		(* Method outputs *)
		(* Clear output data area *)
		(* Number of output arguments *)
		nNoOfOutputArgs := stRemovePathData.iNoOfOutputArgs;
		(* Set up output argument information *)
		MEMSET(ADR(aOutputArgInfo), 0, SIZEOF(aOutputArgInfo));
		aOutputArgInfo[1].DataType := eUAType_Uint16;
		aOutputArgInfo[1].ValueRank := -1;
		aOutputArgInfo[1].nLenData := SIZEOF(stRemovePathData.stOutput.eStatus);
		aOutputArgInfo[2].DataType := eUAType_String;
		aOutputArgInfo[2].ValueRank := -1;
		aOutputArgInfo[2].nLenData := SIZEOF(stRemovePathData.stOutput.sMessage);
		(* Set up output  *)
		MEMSET(ADR(stRemovePathData.stOutput), 0, SIZEOF(stRemovePathData.stOutput));
		stRemovePathData.stOutput.nNumberOfOutputArguments := nNoOfOutputArgs;
		stRemovePathData.stOutput.stOutputArgInfo[1] := aOutputArgInfo[1];
		stRemovePathData.stOutput.stOutputArgInfo[2] := aOutputArgInfo[2];
	
		(* Execute FB *)
		fbCallMethod.nNumberOfInputArguments := nNoOfInputArgs;
		fbCallMethod.pInputArgInfo := ADR(aInputArgInfo);
		fbCallMethod.cbInputArgInfo := (SIZEOF(aInputArgInfo[1])*nNoOfInputArgs);
		fbCallMethod.pInputArgData := ADR(aInputData);
		fbCallMethod.cbInputArgData := nOffset;
		fbCallMethod.nNumberOfOutputArguments := nNoOfOutputArgs; 
		fbCallMethod.pOutputArgInfo := ADR(aOutputArgInfo); 
		fbCallMethod.cbOutputArgInfo := (SIZEOF(aOutputArgInfo[1]) * nNoOfOutputArgs); 
		fbCallMethod.pOutputArgInfoAndData := ADR(stRemovePathData.stOutput);
		fbCallMethod.cbOutputArgInfoAndData := SIZEOF(stRemovePathData.stOutput);
		
		stRemovePathData.iStatus := 1;
		bCallMethod := TRUE;
		
	ELSIF (stRemovePathData.iStatus = 1) THEN
		// Method call Completed...
		IF (eStateMethod = E_TrackClientState.Connected) THEN
			// Method call OK
			IF (stRemovePathData.stOutput.eStatus = E_MMServerStatus.eMMServerStatus_Success) THEN
				// Method returned OK
				stRemovePathData.iStatus := 2;
			ELSE
				// Method returned with error
				stRemovePathData.iStatus := 3;
				stRemovePathData.stOutput.sMessage;
			END_IF
		ELSIF (eStateMethod = E_TrackClientState.Error) THEN
			// Method call failed
			stRemovePathData.iStatus := 3;
		END_IF
		
	END_IF
END_IF

M_CallRemovePath := stRemovePathData.iStatus;
END_METHOD

METHOD PROTECTED M_CallRemovePathSegment : INT
VAR_INPUT
	iSegmentNo		: UINT;
END_VAR
IF (stRemovePathSegmentData.iStatus = 2) OR (stRemovePathSegmentData.iStatus = 3) THEN
	stRemovePathSegmentData.iStatus := 0;
END_IF

IF (bConnectedMethod AND NOT bBusyMethod) THEN
	IF (stRemovePathSegmentData.iStatus = 0) THEN
	(* Setup method calling parameters *)
		(* Method identifier *)
		sObjectIDentifier := stRemovePathSegmentData.sObjectID;
		sMethodIdentifier := stRemovePathSegmentData.sMethodID;
	
		(* Method Inputs *)
		stRemovePathSegmentData.stInput.sCellID := sCellID;
		stRemovePathSegmentData.stInput.sSegmentID := CONCAT(sCellID, '_PS');
		stRemovePathSegmentData.stInput.sSegmentID := CONCAT(stRemovePathSegmentData.stInput.sSegmentID, UINT_TO_STRING(iSegmentNo));			
		(* Fill input data area with method arguments *)
		MEMSET(ADR(aInputData), 0 ,SIZEOF(aInputData));
		nOffset := 0;
		nOffset := nOffset + MEMCPY(ADR(aInputData)+nOffset, ADR(stRemovePathSegmentData.stInput),	MIN(SIZEOF(stRemovePathSegmentData.stInput), (SIZEOF(aInputData)-nOffset)) );
		(* Number of input arguments *)
		nNoOfInputArgs := stRemovePathSegmentData.iNoOfInputArgs;
		(* Set up input argument information *)
		MEMSET(ADR(aInputArgInfo), 0, SIZEOF(aInputArgInfo));
		aInputArgInfo[1].DataType := eUAType_String;
		aInputArgInfo[1].ValueRank := -1;	// -1: Scalar 
		aInputArgInfo[1].nLenData := SIZEOF(stRemovePathSegmentData.stInput.sCellID);
		aInputArgInfo[2].DataType := eUAType_String;
		aInputArgInfo[2].ValueRank := -1;	// -1: Scalar 
		aInputArgInfo[2].nLenData := SIZEOF(stRemovePathSegmentData.stInput.sSegmentID);
		
		(* Method outputs *)
		(* Clear output data area *)
		(* Number of output arguments *)
		nNoOfOutputArgs := stRemovePathSegmentData.iNoOfOutputArgs;
		(* Set up output argument information *)
		MEMSET(ADR(aOutputArgInfo), 0, SIZEOF(aOutputArgInfo));
		aOutputArgInfo[1].DataType := eUAType_Uint16;
		aOutputArgInfo[1].ValueRank := -1;
		aOutputArgInfo[1].nLenData := SIZEOF(stRemovePathSegmentData.stOutput.eStatus);
		aOutputArgInfo[2].DataType := eUAType_String;
		aOutputArgInfo[2].ValueRank := -1;
		aOutputArgInfo[2].nLenData := SIZEOF(stRemovePathSegmentData.stOutput.sMessage);
		(* Set up output  *)
		MEMSET(ADR(stRemovePathSegmentData.stOutput), 0, SIZEOF(stRemovePathSegmentData.stOutput));
		stRemovePathSegmentData.stOutput.nNumberOfOutputArguments := nNoOfOutputArgs;
		stRemovePathSegmentData.stOutput.stOutputArgInfo[1] := aOutputArgInfo[1];
		stRemovePathSegmentData.stOutput.stOutputArgInfo[2] := aOutputArgInfo[2];
	
		(* Execute FB *)
		fbCallMethod.nNumberOfInputArguments := nNoOfInputArgs;
		fbCallMethod.pInputArgInfo := ADR(aInputArgInfo);
		fbCallMethod.cbInputArgInfo := (SIZEOF(aInputArgInfo[1])*nNoOfInputArgs);
		fbCallMethod.pInputArgData := ADR(aInputData);
		fbCallMethod.cbInputArgData := nOffset;
		fbCallMethod.nNumberOfOutputArguments := nNoOfOutputArgs; 
		fbCallMethod.pOutputArgInfo := ADR(aOutputArgInfo); 
		fbCallMethod.cbOutputArgInfo := (SIZEOF(aOutputArgInfo[1]) * nNoOfOutputArgs); 
		fbCallMethod.pOutputArgInfoAndData := ADR(stRemovePathSegmentData.stOutput);
		fbCallMethod.cbOutputArgInfoAndData := SIZEOF(stRemovePathSegmentData.stOutput);
		
		stRemovePathSegmentData.iStatus := 1;
		bCallMethod := TRUE;
		
	ELSIF (stRemovePathSegmentData.iStatus = 1) THEN
		// Method call Completed...
		IF (eStateMethod = E_TrackClientState.Connected) THEN
			// Method call OK
			IF (stRemovePathSegmentData.stOutput.eStatus = E_MMServerStatus.eMMServerStatus_Success) THEN
				// Method returned OK
				stRemovePathSegmentData.iStatus := 2;
			ELSE
				// Method returned with error
				stRemovePathSegmentData.iStatus := 3;
				stRemovePathSegmentData.stOutput.sMessage;
			END_IF
		ELSIF (eStateMethod = E_TrackClientState.Error) THEN
			// Method call failed
			stRemovePathSegmentData.iStatus := 3;
		END_IF
		
	END_IF
END_IF

M_CallRemovePathSegment := stRemovePathSegmentData.iStatus;
END_METHOD

METHOD PROTECTED M_CallRemoveReservation : INT
VAR_INPUT
	sStationID					: STRING(30);												(* The identifier for the station. *)
	nTicket						: UINT;														(*  *)
END_VAR
VAR
	i					: UINT;	
END_VAR
IF (stRemoveReservationData.iStatus = 2) OR (stRemoveReservationData.iStatus = 3) THEN
	stRemoveReservationData.iStatus := 0;
END_IF

IF (bConnectedMethod AND NOT bBusyMethod) THEN
	IF (stRemoveReservationData.iStatus = 0) THEN
	(* Setup method calling parameters *)
		(* Method identifier *)
		sObjectIDentifier := stRemoveReservationData.sObjectID;
		sMethodIdentifier := stRemoveReservationData.sMethodID;
	
		(* Method Inputs *)
		stRemoveReservationData.stInput.sStationID := sStationID;
		stRemoveReservationData.stInput.nTicket := nTicket;
		(* Fill input data area with method arguments *)
		MEMSET(ADR(aInputData), 0 ,SIZEOF(aInputData));
		nOffset := 0;
		nOffset := nOffset + MEMCPY(ADR(aInputData)+nOffset, ADR(stRemoveReservationData.stInput),	MIN(SIZEOF(stRemoveReservationData.stInput), (SIZEOF(aInputData)-nOffset)) );
		(* Number of input arguments *)
		nNoOfInputArgs := stRemoveReservationData.iNoOfInputArgs;
		(* Set up input argument information *)
		MEMSET(ADR(aInputArgInfo), 0, SIZEOF(aInputArgInfo));
		aInputArgInfo[1].DataType := eUAType_String;
		aInputArgInfo[1].ValueRank := -1;	// -1: Scalar 
		aInputArgInfo[1].nLenData := SIZEOF(stRemoveReservationData.stInput.sStationID);
		aInputArgInfo[2].DataType := eUAType_UInt16;
		aInputArgInfo[2].ValueRank := -1;	// -1: Scalar 
		aInputArgInfo[2].nLenData := SIZEOF(stRemoveReservationData.stInput.nTicket);
		
		(* Method outputs *)
		(* Clear output data area *)
		(* Number of output arguments *)
		nNoOfOutputArgs := stRemoveReservationData.iNoOfOutputArgs;
		(* Set up output argument information *)
		MEMSET(ADR(aOutputArgInfo), 0, SIZEOF(aOutputArgInfo));
		aOutputArgInfo[1].DataType := eUAType_Uint16;
		aOutputArgInfo[1].ValueRank := -1;
		aOutputArgInfo[1].nLenData := SIZEOF(stRemoveReservationData.stOutput.eStatus);
		aOutputArgInfo[2].DataType := eUAType_String;
		aOutputArgInfo[2].ValueRank := -1;
		aOutputArgInfo[2].nLenData := SIZEOF(stRemoveReservationData.stOutput.sMessage);
		(* Set up output  *)
		MEMSET(ADR(stRemoveReservationData.stOutput), 0, SIZEOF(stRemoveReservationData.stOutput));
		stRemoveReservationData.stOutput.nNumberOfOutputArguments := nNoOfOutputArgs;
		stRemoveReservationData.stOutput.stOutputArgInfo[1] := aOutputArgInfo[1];
		stRemoveReservationData.stOutput.stOutputArgInfo[2] := aOutputArgInfo[2];
	
		(* Execute FB *)
		fbCallMethod.nNumberOfInputArguments := nNoOfInputArgs;
		fbCallMethod.pInputArgInfo := ADR(aInputArgInfo);
		fbCallMethod.cbInputArgInfo := (SIZEOF(aInputArgInfo[1])*nNoOfInputArgs);
		fbCallMethod.pInputArgData := ADR(aInputData);
		fbCallMethod.cbInputArgData := nOffset;
		fbCallMethod.nNumberOfOutputArguments := nNoOfOutputArgs; 
		fbCallMethod.pOutputArgInfo := ADR(aOutputArgInfo); 
		fbCallMethod.cbOutputArgInfo := (SIZEOF(aOutputArgInfo[1]) * nNoOfOutputArgs); 
		fbCallMethod.pOutputArgInfoAndData := ADR(stRemoveReservationData.stOutput);
		fbCallMethod.cbOutputArgInfoAndData := SIZEOF(stRemoveReservationData.stOutput);
		
		stRemoveReservationData.iStatus := 1;
		bCallMethod := TRUE;
		
	ELSIF (stRemoveReservationData.iStatus = 1) THEN
		// Method call Completed...
		IF (eStateMethod = E_TrackClientState.Connected) THEN
			// Method call OK
			IF (stRemoveReservationData.stOutput.eStatus = E_MMServerStatus.eMMServerStatus_Success) THEN
				// Method returned OK
				stRemoveReservationData.iStatus := 2;
			ELSE
				// Method returned with error
				stRemoveReservationData.iStatus := 3;
				stRemoveReservationData.stOutput.sMessage;
			END_IF
		ELSIF (eStateMethod = E_TrackClientState.Error) THEN
			// Method call failed
			stRemoveReservationData.iStatus := 3;
		END_IF
		
	END_IF
END_IF

M_CallRemoveReservation := stRemoveReservationData.iStatus;
END_METHOD

METHOD PROTECTED M_CallRemoveStation : INT
VAR_INPUT
	nStationNo			: UINT(1..5);
END_VAR
IF (stRemoveStationData.iStatus = 2) OR (stRemoveStationData.iStatus = 3) THEN
	stRemoveStationData.iStatus := 0;
END_IF

IF (bConnectedMethod AND NOT bBusyMethod) THEN
	IF (stRemoveStationData.iStatus = 0) THEN
	(* Setup method calling parameters *)
		(* Method identifier *)
		sObjectIDentifier := stRemoveStationData.sObjectID;
		sMethodIdentifier := stRemoveStationData.sMethodID;
	
		(* Method Inputs *)
		stRemoveStationData.stInput.sCellID := sCellID;
		stRemoveStationData.stInput.sStationID := aStations[nStationNo].sStationID;
		(* Fill input data area with method arguments *)
		MEMSET(ADR(aInputData), 0 ,SIZEOF(aInputData));
		nOffset := 0;
		nOffset := nOffset + MEMCPY(ADR(aInputData)+nOffset, ADR(stRemoveStationData.stInput),	MIN(SIZEOF(stRemoveStationData.stInput), (SIZEOF(aInputData)-nOffset)) );
		(* Number of input arguments *)
		nNoOfInputArgs := stRemoveStationData.iNoOfInputArgs;
		(* Set up input argument information *)
		MEMSET(ADR(aInputArgInfo), 0, SIZEOF(aInputArgInfo));
		aInputArgInfo[1].DataType := eUAType_String;
		aInputArgInfo[1].ValueRank := -1;	// -1: Scalar 
		aInputArgInfo[1].nLenData := SIZEOF(stRemoveStationData.stInput.sCellID);
		aInputArgInfo[2].DataType := eUAType_String;
		aInputArgInfo[2].ValueRank := -1;	// -1: Scalar 
		aInputArgInfo[2].nLenData := SIZEOF(stRemoveStationData.stInput.sStationID);
		
		(* Method outputs *)
		(* Clear output data area *)
		(* Number of output arguments *)
		nNoOfOutputArgs := stRemoveStationData.iNoOfOutputArgs;
		(* Set up output argument information *)
		MEMSET(ADR(aOutputArgInfo), 0, SIZEOF(aOutputArgInfo));
		aOutputArgInfo[1].DataType := eUAType_Uint16;
		aOutputArgInfo[1].ValueRank := -1;
		aOutputArgInfo[1].nLenData := SIZEOF(stRemoveStationData.stOutput.eStatus);
		aOutputArgInfo[2].DataType := eUAType_String;
		aOutputArgInfo[2].ValueRank := -1;
		aOutputArgInfo[2].nLenData := SIZEOF(stRemoveStationData.stOutput.sMessage);
		(* Set up output  *)
		MEMSET(ADR(stRemoveStationData.stOutput), 0, SIZEOF(stRemoveStationData.stOutput));
		stRemoveStationData.stOutput.nNumberOfOutputArguments := nNoOfOutputArgs;
		stRemoveStationData.stOutput.stOutputArgInfo[1] := aOutputArgInfo[1];
		stRemoveStationData.stOutput.stOutputArgInfo[2] := aOutputArgInfo[2];
	
		(* Execute FB *)
		fbCallMethod.nNumberOfInputArguments := nNoOfInputArgs;
		fbCallMethod.pInputArgInfo := ADR(aInputArgInfo);
		fbCallMethod.cbInputArgInfo := (SIZEOF(aInputArgInfo[1])*nNoOfInputArgs);
		fbCallMethod.pInputArgData := ADR(aInputData);
		fbCallMethod.cbInputArgData := nOffset;
		fbCallMethod.nNumberOfOutputArguments := nNoOfOutputArgs; 
		fbCallMethod.pOutputArgInfo := ADR(aOutputArgInfo); 
		fbCallMethod.cbOutputArgInfo := (SIZEOF(aOutputArgInfo[1]) * nNoOfOutputArgs); 
		fbCallMethod.pOutputArgInfoAndData := ADR(stRemoveStationData.stOutput);
		fbCallMethod.cbOutputArgInfoAndData := SIZEOF(stRemoveStationData.stOutput);
		
		stRemoveStationData.iStatus := 1;
		bCallMethod := TRUE;
		
	ELSIF (stRemoveStationData.iStatus = 1) THEN
		// Method call Completed...
		IF (eStateMethod = E_TrackClientState.Connected) THEN
			// Method call OK
			IF (stRemoveStationData.stOutput.eStatus = E_MMServerStatus.eMMServerStatus_Success) THEN
				// Method returned OK
				stRemoveStationData.iStatus := 2;
			ELSE
				// Method returned with error
				stRemoveStationData.iStatus := 3;
				stRemoveStationData.stOutput.sMessage;
			END_IF
		ELSIF (eStateMethod = E_TrackClientState.Error) THEN
			// Method call failed
			stRemoveStationData.iStatus := 3;
		END_IF
		
	END_IF
END_IF

M_CallRemoveStation := stRemoveStationData.iStatus;
END_METHOD

METHOD PROTECTED M_CallRemoveTrafficLight : INT
VAR_INPUT
END_VAR
IF (stRemoveTrafficLightData.iStatus = 2) OR (stRemoveTrafficLightData.iStatus = 3) THEN
	stRemoveTrafficLightData.iStatus := 0;
END_IF

IF (bConnectedMethod AND NOT bBusyMethod) THEN
	IF (stRemoveTrafficLightData.iStatus = 0) THEN
	(* Setup method calling parameters *)
		(* Method identifier *)
		sObjectIDentifier := stRemoveTrafficLightData.sObjectID;
		sMethodIdentifier := stRemoveTrafficLightData.sMethodID;
	
		(* Method Inputs *)
		stRemoveTrafficLightData.stInput.sCellID := sCellID;
		stRemoveTrafficLightData.stInput.sID := CONCAT(sCellID, '_TL');
		(* Fill input data area with method arguments *)
		MEMSET(ADR(aInputData), 0 ,SIZEOF(aInputData));
		nOffset := 0;
		nOffset := nOffset + MEMCPY(ADR(aInputData)+nOffset, ADR(stRemoveTrafficLightData.stInput),	MIN(SIZEOF(stRemoveTrafficLightData.stInput),	(SIZEOF(aInputData)-nOffset)) );
		(* Number of input arguments *)
		nNoOfInputArgs := stRemoveTrafficLightData.iNoOfInputArgs;
		(* Set up input argument information *)
		MEMSET(ADR(aInputArgInfo), 0, SIZEOF(aInputArgInfo));
		aInputArgInfo[1].DataType := eUAType_String;
		aInputArgInfo[1].ValueRank := -1;	// -1: Scalar 
		aInputArgInfo[1].nLenData := SIZEOF(stRemoveTrafficLightData.stInput.sCellID);
		aInputArgInfo[2].DataType := eUAType_String;
		aInputArgInfo[2].ValueRank := -1;	// -1: Scalar 
		aInputArgInfo[2].nLenData := SIZEOF(stRemoveTrafficLightData.stInput.sID);
		
		(* Method outputs *)
		(* Clear output data area *)
		(* Number of output arguments *)
		nNoOfOutputArgs := stRemoveTrafficLightData.iNoOfOutputArgs;
		(* Set up output argument information *)
		MEMSET(ADR(aOutputArgInfo), 0, SIZEOF(aOutputArgInfo));
		aOutputArgInfo[1].DataType := eUAType_Uint16;
		aOutputArgInfo[1].ValueRank := -1;
		aOutputArgInfo[1].nLenData := SIZEOF(stRemoveTrafficLightData.stOutput.eStatus);
		aOutputArgInfo[2].DataType := eUAType_String;
		aOutputArgInfo[2].ValueRank := -1;
		aOutputArgInfo[2].nLenData := SIZEOF(stRemoveTrafficLightData.stOutput.sMessage);
		(* Set up output  *)
		MEMSET(ADR(stRemoveTrafficLightData.stOutput), 0, SIZEOF(stRemoveTrafficLightData.stOutput));
		stRemoveTrafficLightData.stOutput.nNumberOfOutputArguments := nNoOfOutputArgs;
		stRemoveTrafficLightData.stOutput.stOutputArgInfo[1] := aOutputArgInfo[1];
		stRemoveTrafficLightData.stOutput.stOutputArgInfo[2] := aOutputArgInfo[2];
	
		(* Execute FB *)
		fbCallMethod.nNumberOfInputArguments := nNoOfInputArgs;
		fbCallMethod.pInputArgInfo := ADR(aInputArgInfo);
		fbCallMethod.cbInputArgInfo := (SIZEOF(aInputArgInfo[1])*nNoOfInputArgs);
		fbCallMethod.pInputArgData := ADR(aInputData);
		fbCallMethod.cbInputArgData := nOffset;
		fbCallMethod.nNumberOfOutputArguments := nNoOfOutputArgs; 
		fbCallMethod.pOutputArgInfo := ADR(aOutputArgInfo); 
		fbCallMethod.cbOutputArgInfo := (SIZEOF(aOutputArgInfo[1]) * nNoOfOutputArgs); 
		fbCallMethod.pOutputArgInfoAndData := ADR(stRemoveTrafficLightData.stOutput);
		fbCallMethod.cbOutputArgInfoAndData := SIZEOF(stRemoveTrafficLightData.stOutput);
		
		stRemoveTrafficLightData.iStatus := 1;
		bCallMethod := TRUE;
		
	ELSIF (stRemoveTrafficLightData.iStatus = 1) THEN
		// Method call Completed...
		IF (eStateMethod = E_TrackClientState.Connected) THEN
			// Method call OK
			IF (stRemoveTrafficLightData.stOutput.eStatus = E_MMServerStatus.eMMServerStatus_Success) THEN
				// Method returned OK
				stRemoveTrafficLightData.iStatus := 2;
			ELSE
				// Method returned with error
				stRemoveTrafficLightData.iStatus := 3;
				stRemoveTrafficLightData.stOutput.sMessage;
			END_IF
		ELSIF (eStateMethod = E_TrackClientState.Error) THEN
			// Method call failed
			stRemoveTrafficLightData.iStatus := 3;
		END_IF
		
	END_IF
END_IF

M_CallRemoveTrafficLight := stRemoveTrafficLightData.iStatus;
END_METHOD

METHOD PROTECTED M_CallResetPath : INT
VAR_INPUT
	nPathNo			: UINT(1..5);
END_VAR
IF (stResetPathData.iStatus = 2) OR (stResetPathData.iStatus = 3) THEN
	stResetPathData.iStatus := 0;
END_IF

IF (bConnectedMethod AND NOT bBusyMethod) THEN
	IF (stResetPathData.iStatus = 0) THEN
	(* Setup method calling parameters *)
		(* Method identifier *)
		sObjectIDentifier := stResetPathData.sObjectID;
		sMethodIdentifier := stResetPathData.sMethodID;
	
		(* Method Inputs *)
		stResetPathData.stInput.iPath := nPathNo;
		(* Fill input data area with method arguments *)
		MEMSET(ADR(aInputData), 0 ,SIZEOF(aInputData));
		nOffset := 0;
		nOffset := nOffset + MEMCPY(ADR(aInputData)+nOffset, ADR(stResetPathData.stInput),	MIN(SIZEOF(stResetPathData.stInput), (SIZEOF(aInputData)-nOffset)) );
		(* Number of input arguments *)
		nNoOfInputArgs := stResetPathData.iNoOfInputArgs;
		(* Set up input argument information *)
		MEMSET(ADR(aInputArgInfo), 0, SIZEOF(aInputArgInfo));
		aInputArgInfo[1].DataType := eUAType_UInt16;
		aInputArgInfo[1].ValueRank := -1;	// -1: Scalar 
		aInputArgInfo[1].nLenData := SIZEOF(stResetPathData.stInput.iPath);
		
		(* Method outputs *)
		(* Clear output data area *)
		(* Number of output arguments *)
		nNoOfOutputArgs := stResetPathData.iNoOfOutputArgs;
		(* Set up output argument information *)
		MEMSET(ADR(aOutputArgInfo), 0, SIZEOF(aOutputArgInfo));
		aOutputArgInfo[1].DataType := eUAType_Uint16;
		aOutputArgInfo[1].ValueRank := -1;
		aOutputArgInfo[1].nLenData := SIZEOF(stResetPathData.stOutput.eStatus);
		aOutputArgInfo[2].DataType := eUAType_String;
		aOutputArgInfo[2].ValueRank := -1;
		aOutputArgInfo[2].nLenData := SIZEOF(stResetPathData.stOutput.sMessage);
		(* Set up output  *)
		MEMSET(ADR(stResetPathData.stOutput), 0, SIZEOF(stResetPathData.stOutput));
		stResetPathData.stOutput.nNumberOfOutputArguments := nNoOfOutputArgs;
		stResetPathData.stOutput.stOutputArgInfo[1] := aOutputArgInfo[1];
		stResetPathData.stOutput.stOutputArgInfo[2] := aOutputArgInfo[2];
	
		(* Execute FB *)
		fbCallMethod.nNumberOfInputArguments := nNoOfInputArgs;
		fbCallMethod.pInputArgInfo := ADR(aInputArgInfo);
		fbCallMethod.cbInputArgInfo := (SIZEOF(aInputArgInfo[1])*nNoOfInputArgs);
		fbCallMethod.pInputArgData := ADR(aInputData);
		fbCallMethod.cbInputArgData := nOffset;
		fbCallMethod.nNumberOfOutputArguments := nNoOfOutputArgs; 
		fbCallMethod.pOutputArgInfo := ADR(aOutputArgInfo); 
		fbCallMethod.cbOutputArgInfo := (SIZEOF(aOutputArgInfo[1]) * nNoOfOutputArgs); 
		fbCallMethod.pOutputArgInfoAndData := ADR(stResetPathData.stOutput);
		fbCallMethod.cbOutputArgInfoAndData := SIZEOF(stResetPathData.stOutput);
		
		stResetPathData.iStatus := 1;
		bCallMethod := TRUE;
		
	ELSIF (stResetPathData.iStatus = 1) THEN
		// Method call Completed...
		IF (eStateMethod = E_TrackClientState.Connected) THEN
			// eStateMethod call OK
			IF (stResetPathData.stOutput.eStatus = E_MMServerStatus.eMMServerStatus_Success) THEN
				// Method returned OK
				stResetPathData.iStatus := 2;
			ELSE
				// Method returned with error
				stResetPathData.iStatus := 3;
				stResetPathData.stOutput.sMessage;
			END_IF
		ELSIF (eStateMethod = E_TrackClientState.Error) THEN
			// Method call failed
			stResetPathData.iStatus := 3;
		END_IF
		
	END_IF
END_IF

M_CallResetPath := stResetPathData.iStatus;
END_METHOD

METHOD PROTECTED M_CallResumePath : INT
VAR_INPUT
	nPathNo			: UINT(1..5);
END_VAR
IF (stResumePathData.iStatus = 2) OR (stResumePathData.iStatus = 3) THEN
	stResumePathData.iStatus := 0;
END_IF

IF (bConnectedMethod AND NOT bBusyMethod) THEN
	IF (stResumePathData.iStatus = 0) THEN
	(* Setup method calling parameters *)
		(* Method identifier *)
		sObjectIDentifier := stResumePathData.sObjectID;
		sMethodIdentifier := stResumePathData.sMethodID;
	
		(* Method Inputs *)
		stResumePathData.stInput.iPath := nPathNo;
		(* Fill input data area with method arguments *)
		MEMSET(ADR(aInputData), 0 ,SIZEOF(aInputData));
		nOffset := 0;
		nOffset := nOffset + MEMCPY(ADR(aInputData)+nOffset, ADR(stResumePathData.stInput),	MIN(SIZEOF(stResumePathData.stInput), (SIZEOF(aInputData)-nOffset)) );
		(* Number of input arguments *)
		nNoOfInputArgs := stResumePathData.iNoOfInputArgs;
		(* Set up input argument information *)
		MEMSET(ADR(aInputArgInfo), 0, SIZEOF(aInputArgInfo));
		aInputArgInfo[1].DataType := eUAType_UInt16;
		aInputArgInfo[1].ValueRank := -1;	// -1: Scalar 
		aInputArgInfo[1].nLenData := SIZEOF(stResumePathData.stInput.iPath);
		
		(* Method outputs *)
		(* Clear output data area *)
		(* Number of output arguments *)
		nNoOfOutputArgs := stResumePathData.iNoOfOutputArgs;
		(* Set up output argument information *)
		MEMSET(ADR(aOutputArgInfo), 0, SIZEOF(aOutputArgInfo));
		aOutputArgInfo[1].DataType := eUAType_Uint16;
		aOutputArgInfo[1].ValueRank := -1;
		aOutputArgInfo[1].nLenData := SIZEOF(stResumePathData.stOutput.eStatus);
		aOutputArgInfo[2].DataType := eUAType_String;
		aOutputArgInfo[2].ValueRank := -1;
		aOutputArgInfo[2].nLenData := SIZEOF(stResumePathData.stOutput.sMessage);
		(* Set up output  *)
		MEMSET(ADR(stResumePathData.stOutput), 0, SIZEOF(stResumePathData.stOutput));
		stResumePathData.stOutput.nNumberOfOutputArguments := nNoOfOutputArgs;
		stResumePathData.stOutput.stOutputArgInfo[1] := aOutputArgInfo[1];
		stResumePathData.stOutput.stOutputArgInfo[2] := aOutputArgInfo[2];
	
		(* Execute FB *)
		fbCallMethod.nNumberOfInputArguments := nNoOfInputArgs;
		fbCallMethod.pInputArgInfo := ADR(aInputArgInfo);
		fbCallMethod.cbInputArgInfo := (SIZEOF(aInputArgInfo[1])*nNoOfInputArgs);
		fbCallMethod.pInputArgData := ADR(aInputData);
		fbCallMethod.cbInputArgData := nOffset;
		fbCallMethod.nNumberOfOutputArguments := nNoOfOutputArgs; 
		fbCallMethod.pOutputArgInfo := ADR(aOutputArgInfo); 
		fbCallMethod.cbOutputArgInfo := (SIZEOF(aOutputArgInfo[1]) * nNoOfOutputArgs); 
		fbCallMethod.pOutputArgInfoAndData := ADR(stResumePathData.stOutput);
		fbCallMethod.cbOutputArgInfoAndData := SIZEOF(stResumePathData.stOutput);
		
		stResumePathData.iStatus := 1;
		bCallMethod := TRUE;
		
	ELSIF (stResumePathData.iStatus = 1) THEN
		// Method call Completed...
		IF (eStateMethod = E_TrackClientState.Connected) THEN
			// Method call OK
			IF (stResumePathData.stOutput.eStatus = E_MMServerStatus.eMMServerStatus_Success) THEN
				// Method returned OK
				stResumePathData.iStatus := 2;
			ELSE
				// Method returned with error
				stResumePathData.iStatus := 3;
				stResumePathData.stOutput.sMessage;
			END_IF
		ELSIF (eStateMethod = E_TrackClientState.Error) THEN
			// Method call failed
			stResumePathData.iStatus := 3;
		END_IF
		
	END_IF
END_IF

M_CallResumePath := stResumePathData.iStatus;
END_METHOD

METHOD PROTECTED M_CallSetTrafficLightColor : INT
VAR_INPUT
	nTrafficLightNo	: UINT;
	nColor			: INT;
END_VAR
IF (stSetTrafficLightColorData.iStatus = 2) OR (stSetTrafficLightColorData.iStatus = 3) THEN
	stSetTrafficLightColorData.iStatus := 0;
END_IF

IF (bConnectedMethod AND NOT bBusyMethod) THEN
	IF (stSetTrafficLightColorData.iStatus = 0) THEN
	(* Setup method calling parameters *)
		(* Method identifier *)
		sObjectIDentifier := stSetTrafficLightColorData.sObjectID;
		sMethodIdentifier := stSetTrafficLightColorData.sMethodID;
			
		(* Method Inputs *)
		stSetTrafficLightColorData.stInput.sCellID := sCellID;
		stSetTrafficLightColorData.stInput.sID := CONCAT(sCellID, '_TL');
		stSetTrafficLightColorData.stInput.sID := CONCAT(stSetTrafficLightColorData.stInput.sID, UINT_TO_STRING(nTrafficLightNo));
		stSetTrafficLightColorData.stInput.nColor := nColor;
		(* Fill input data area with method arguments *)
		MEMSET(ADR(aInputData), 0 ,SIZEOF(aInputData));
		nOffset := 0;
		nOffset := nOffset + MEMCPY(ADR(aInputData)+nOffset, ADR(stSetTrafficLightColorData.stInput),	MIN(SIZEOF(stSetTrafficLightColorData.stInput),	(SIZEOF(aInputData)-nOffset)) );
		(* Number of input arguments *)
		nNoOfInputArgs := stSetTrafficLightColorData.iNoOfInputArgs;
		(* Set up input argument information *)
		MEMSET(ADR(aInputArgInfo), 0, SIZEOF(aInputArgInfo));
		aInputArgInfo[1].DataType := eUAType_String;
		aInputArgInfo[1].ValueRank := -1;	// -1: Scalar 
		aInputArgInfo[1].nLenData := SIZEOF(stSetTrafficLightColorData.stInput.sCellID);
		aInputArgInfo[2].DataType := eUAType_String;
		aInputArgInfo[2].ValueRank := -1;	// -1: Scalar 
		aInputArgInfo[2].nLenData := SIZEOF(stSetTrafficLightColorData.stInput.sID);
		aInputArgInfo[3].DataType := eUAType_Int16;
		aInputArgInfo[3].ValueRank := -1;	// -1: Scalar 
		aInputArgInfo[3].nLenData := SIZEOF(nColor);
		
		(* Method outputs *)
		(* Clear output data area *)
		(* Number of output arguments *)
		nNoOfOutputArgs := stSetTrafficLightColorData.iNoOfOutputArgs;
		(* Set up output argument information *)
		MEMSET(ADR(aOutputArgInfo), 0, SIZEOF(aOutputArgInfo));
		aOutputArgInfo[1].DataType := eUAType_Uint16;
		aOutputArgInfo[1].ValueRank := -1;
		aOutputArgInfo[1].nLenData := SIZEOF(stSetTrafficLightColorData.stOutput.eStatus);
		aOutputArgInfo[2].DataType := eUAType_String;
		aOutputArgInfo[2].ValueRank := -1;
		aOutputArgInfo[2].nLenData := SIZEOF(stSetTrafficLightColorData.stOutput.sMessage);
		(* Set up output  *)
		MEMSET(ADR(stSetTrafficLightColorData.stOutput), 0, SIZEOF(stSetTrafficLightColorData.stOutput));
		stSetTrafficLightColorData.stOutput.nNumberOfOutputArguments := nNoOfOutputArgs;
		stSetTrafficLightColorData.stOutput.stOutputArgInfo[1] := aOutputArgInfo[1];
		stSetTrafficLightColorData.stOutput.stOutputArgInfo[2] := aOutputArgInfo[2];
	
		(* Execute FB *)
		fbCallMethod.nNumberOfInputArguments := nNoOfInputArgs;
		fbCallMethod.pInputArgInfo := ADR(aInputArgInfo);
		fbCallMethod.cbInputArgInfo := (SIZEOF(aInputArgInfo[1])*nNoOfInputArgs);
		fbCallMethod.pInputArgData := ADR(aInputData);
		fbCallMethod.cbInputArgData := nOffset;
		fbCallMethod.nNumberOfOutputArguments := nNoOfOutputArgs; 
		fbCallMethod.pOutputArgInfo := ADR(aOutputArgInfo); 
		fbCallMethod.cbOutputArgInfo := (SIZEOF(aOutputArgInfo[1]) * nNoOfOutputArgs); 
		fbCallMethod.pOutputArgInfoAndData := ADR(stSetTrafficLightColorData.stOutput);
		fbCallMethod.cbOutputArgInfoAndData := SIZEOF(stSetTrafficLightColorData.stOutput);
		
		stSetTrafficLightColorData.iStatus := 1;
		bCallMethod := TRUE;
		
	ELSIF (stSetTrafficLightColorData.iStatus = 1) THEN
		// Method call Completed...
		IF (eStateMethod = E_TrackClientState.Connected) THEN
			// Method call OK
			IF (stSetTrafficLightColorData.stOutput.eStatus = E_MMServerStatus.eMMServerStatus_Success) THEN
				// Method returned OK
				stSetTrafficLightColorData.iStatus := 2;
			ELSE
				// Method returned with error
				stSetTrafficLightColorData.iStatus := 3;
				stSetTrafficLightColorData.stOutput.sMessage;
			END_IF
		ELSIF (eStateMethod = E_TrackClientState.Error) THEN
			// Method call failed
			stSetTrafficLightColorData.iStatus := 3;
		END_IF
		
	END_IF
END_IF

M_CallSetTrafficLightColor := stSetTrafficLightColorData.iStatus;
END_METHOD

METHOD PROTECTED M_CallStartPath : INT
VAR_INPUT
	nPathNo			: UINT(1..5);
END_VAR
IF (stStartPathData.iStatus = 2) OR (stStartPathData.iStatus = 3) THEN
	stStartPathData.iStatus := 0;
END_IF

IF (bConnectedMethod AND NOT bBusyMethod) THEN
	IF (stStartPathData.iStatus = 0) THEN
	(* Setup method calling parameters *)
		(* Method identifier *)
		sObjectIDentifier := stStartPathData.sObjectID;
		sMethodIdentifier := stStartPathData.sMethodID;
	
		(* Method Inputs *)
		stStartPathData.stInput.iPath := nPathNo;
		(* Fill input data area with method arguments *)
		MEMSET(ADR(aInputData), 0 ,SIZEOF(aInputData));
		nOffset := 0;
		nOffset := nOffset + MEMCPY(ADR(aInputData)+nOffset, ADR(stStartPathData.stInput),	MIN(SIZEOF(stStartPathData.stInput), (SIZEOF(aInputData)-nOffset)) );
		(* Number of input arguments *)
		nNoOfInputArgs := stStartPathData.iNoOfInputArgs;
		(* Set up input argument information *)
		MEMSET(ADR(aInputArgInfo), 0, SIZEOF(aInputArgInfo));
		aInputArgInfo[1].DataType := eUAType_UInt16;
		aInputArgInfo[1].ValueRank := -1;	// -1: Scalar 
		aInputArgInfo[1].nLenData := SIZEOF(stStartPathData.stInput.iPath);
		
		(* Method outputs *)
		(* Clear output data area *)
		(* Number of output arguments *)
		nNoOfOutputArgs := stStartPathData.iNoOfOutputArgs;
		(* Set up output argument information *)
		MEMSET(ADR(aOutputArgInfo), 0, SIZEOF(aOutputArgInfo));
		aOutputArgInfo[1].DataType := eUAType_Uint16;
		aOutputArgInfo[1].ValueRank := -1;
		aOutputArgInfo[1].nLenData := SIZEOF(stStartPathData.stOutput.eStatus);
		aOutputArgInfo[2].DataType := eUAType_String;
		aOutputArgInfo[2].ValueRank := -1;
		aOutputArgInfo[2].nLenData := SIZEOF(stStartPathData.stOutput.sMessage);
		(* Set up output  *)
		MEMSET(ADR(stStartPathData.stOutput), 0, SIZEOF(stStartPathData.stOutput));
		stStartPathData.stOutput.nNumberOfOutputArguments := nNoOfOutputArgs;
		stStartPathData.stOutput.stOutputArgInfo[1] := aOutputArgInfo[1];
		stStartPathData.stOutput.stOutputArgInfo[2] := aOutputArgInfo[2];
	
		(* Execute FB *)
		fbCallMethod.nNumberOfInputArguments := nNoOfInputArgs;
		fbCallMethod.pInputArgInfo := ADR(aInputArgInfo);
		fbCallMethod.cbInputArgInfo := (SIZEOF(aInputArgInfo[1])*nNoOfInputArgs);
		fbCallMethod.pInputArgData := ADR(aInputData);
		fbCallMethod.cbInputArgData := nOffset;
		fbCallMethod.nNumberOfOutputArguments := nNoOfOutputArgs; 
		fbCallMethod.pOutputArgInfo := ADR(aOutputArgInfo); 
		fbCallMethod.cbOutputArgInfo := (SIZEOF(aOutputArgInfo[1]) * nNoOfOutputArgs); 
		fbCallMethod.pOutputArgInfoAndData := ADR(stStartPathData.stOutput);
		fbCallMethod.cbOutputArgInfoAndData := SIZEOF(stStartPathData.stOutput);
		
		stStartPathData.iStatus := 1;
		bCallMethod := TRUE;
		
	ELSIF (stStartPathData.iStatus = 1) THEN
		// Method call Completed...
		IF (eStateMethod = E_TrackClientState.Connected) THEN
			// Method call OK
			IF (stStartPathData.stOutput.eStatus = E_MMServerStatus.eMMServerStatus_Success) THEN
				// Method returned OK
				stStartPathData.iStatus := 2;
			ELSE
				// Method returned with error
				stStartPathData.iStatus := 3;
				stStartPathData.stOutput.sMessage;
			END_IF
		ELSIF (eStateMethod = E_TrackClientState.Error) THEN
			// Method call failed
			stStartPathData.iStatus := 3;
		END_IF
		
	END_IF
END_IF

M_CallStartPath := stStartPathData.iStatus;
END_METHOD

METHOD PROTECTED M_CallSuspendPath : INT
VAR_INPUT
	nPathNo			: UINT(1..5);
END_VAR
IF (stSuspendPathData.iStatus = 2) OR (stSuspendPathData.iStatus = 3) THEN
	stSuspendPathData.iStatus := 0;
END_IF

IF (bConnectedMethod AND NOT bBusyMethod) THEN
	IF (stSuspendPathData.iStatus = 0) THEN
	(* Setup method calling parameters *)
		(* Method identifier *)
		sObjectIDentifier := stSuspendPathData.sObjectID;
		sMethodIdentifier := stSuspendPathData.sMethodID;
	
		(* Method Inputs *)
		stSuspendPathData.stInput.iPath := nPathNo;
		(* Fill input data area with method arguments *)
		MEMSET(ADR(aInputData), 0 ,SIZEOF(aInputData));
		nOffset := 0;
		nOffset := nOffset + MEMCPY(ADR(aInputData)+nOffset, ADR(stSuspendPathData.stInput),	MIN(SIZEOF(stSuspendPathData.stInput), (SIZEOF(aInputData)-nOffset)) );
		(* Number of input arguments *)
		nNoOfInputArgs := stSuspendPathData.iNoOfInputArgs;
		(* Set up input argument information *)
		MEMSET(ADR(aInputArgInfo), 0, SIZEOF(aInputArgInfo));
		aInputArgInfo[1].DataType := eUAType_UInt16;
		aInputArgInfo[1].ValueRank := -1;	// -1: Scalar 
		aInputArgInfo[1].nLenData := SIZEOF(stSuspendPathData.stInput.iPath);
		
		(* Method outputs *)
		(* Clear output data area *)
		(* Number of output arguments *)
		nNoOfOutputArgs := stSuspendPathData.iNoOfOutputArgs;
		(* Set up output argument information *)
		MEMSET(ADR(aOutputArgInfo), 0, SIZEOF(aOutputArgInfo));
		aOutputArgInfo[1].DataType := eUAType_Uint16;
		aOutputArgInfo[1].ValueRank := -1;
		aOutputArgInfo[1].nLenData := SIZEOF(stSuspendPathData.stOutput.eStatus);
		aOutputArgInfo[2].DataType := eUAType_String;
		aOutputArgInfo[2].ValueRank := -1;
		aOutputArgInfo[2].nLenData := SIZEOF(stSuspendPathData.stOutput.sMessage);
		(* Set up output  *)
		MEMSET(ADR(stSuspendPathData.stOutput), 0, SIZEOF(stSuspendPathData.stOutput));
		stSuspendPathData.stOutput.nNumberOfOutputArguments := nNoOfOutputArgs;
		stSuspendPathData.stOutput.stOutputArgInfo[1] := aOutputArgInfo[1];
		stSuspendPathData.stOutput.stOutputArgInfo[2] := aOutputArgInfo[2];
	
		(* Execute FB *)
		fbCallMethod.nNumberOfInputArguments := nNoOfInputArgs;
		fbCallMethod.pInputArgInfo := ADR(aInputArgInfo);
		fbCallMethod.cbInputArgInfo := (SIZEOF(aInputArgInfo[1])*nNoOfInputArgs);
		fbCallMethod.pInputArgData := ADR(aInputData);
		fbCallMethod.cbInputArgData := nOffset;
		fbCallMethod.nNumberOfOutputArguments := nNoOfOutputArgs; 
		fbCallMethod.pOutputArgInfo := ADR(aOutputArgInfo); 
		fbCallMethod.cbOutputArgInfo := (SIZEOF(aOutputArgInfo[1]) * nNoOfOutputArgs); 
		fbCallMethod.pOutputArgInfoAndData := ADR(stSuspendPathData.stOutput);
		fbCallMethod.cbOutputArgInfoAndData := SIZEOF(stSuspendPathData.stOutput);
		
		stSuspendPathData.iStatus := 1;
		bCallMethod := TRUE;
		
	ELSIF (stSuspendPathData.iStatus = 1) THEN
		// Method call Completed...
		IF (eStateMethod = E_TrackClientState.Connected) THEN
			// Method call OK
			IF (stSuspendPathData.stOutput.eStatus = E_MMServerStatus.eMMServerStatus_Success) THEN
				// Method returned OK
				stSuspendPathData.iStatus := 2;
			ELSE
				// Method returned with error
				stSuspendPathData.iStatus := 3;
				stSuspendPathData.stOutput.sMessage;
			END_IF
		ELSIF (eStateMethod = E_TrackClientState.Error) THEN
			// Method call failed
			stSuspendPathData.iStatus := 3;
		END_IF
		
	END_IF
END_IF

M_CallSuspendPath := stSuspendPathData.iStatus;
END_METHOD

METHOD PROTECTED M_CallTrafficLightColor : INT
VAR_INPUT
END_VAR
IF (stTrafficLightColorData.iStatus = 2) OR (stTrafficLightColorData.iStatus = 3) THEN
	stTrafficLightColorData.iStatus := 0;
END_IF

IF (bConnectedMethod AND NOT bBusyMethod) THEN
	IF (stTrafficLightColorData.iStatus = 0) THEN
	(* Setup method calling parameters *)
		(* Method identifier *)
		sObjectIDentifier := stTrafficLightColorData.sObjectID;
		sMethodIdentifier := stTrafficLightColorData.sMethodID;
	
		(* Method Inputs *)
		stTrafficLightColorData.stInput.sCellID := sCellID;
		stTrafficLightColorData.stInput.sID := CONCAT(sCellID, '_TL');
		(* Fill input data area with method arguments *)
		MEMSET(ADR(aInputData), 0 ,SIZEOF(aInputData));
		nOffset := 0;
		nOffset := nOffset + MEMCPY(ADR(aInputData)+nOffset, ADR(stTrafficLightColorData.stInput),	MIN(SIZEOF(stTrafficLightColorData.stInput), (SIZEOF(aInputData)-nOffset)) );
		(* Number of input arguments *)
		nNoOfInputArgs := stTrafficLightColorData.iNoOfInputArgs;
		(* Set up input argument information *)
		MEMSET(ADR(aInputArgInfo), 0, SIZEOF(aInputArgInfo));
		aInputArgInfo[1].DataType := eUAType_String;
		aInputArgInfo[1].ValueRank := -1;	// -1: Scalar 
		aInputArgInfo[1].nLenData := SIZEOF(stTrafficLightColorData.stInput.sCellID);
		aInputArgInfo[2].DataType := eUAType_String;
		aInputArgInfo[2].ValueRank := -1;	// -1: Scalar 
		aInputArgInfo[2].nLenData := SIZEOF(stTrafficLightColorData.stInput.sID);
		
		(* Method outputs *)
		(* Clear output data area *)
		(* Number of output arguments *)
		nNoOfOutputArgs := stTrafficLightColorData.iNoOfOutputArgs;
		(* Set up output argument information *)
		MEMSET(ADR(aOutputArgInfo), 0, SIZEOF(aOutputArgInfo));
		aOutputArgInfo[1].DataType := eUAType_Uint16;
		aOutputArgInfo[1].ValueRank := -1;
		aOutputArgInfo[1].nLenData := SIZEOF(stTrafficLightColorData.stOutput.eStatus);
		aOutputArgInfo[2].DataType := eUAType_String;
		aOutputArgInfo[2].ValueRank := -1;
		aOutputArgInfo[2].nLenData := SIZEOF(stTrafficLightColorData.stOutput.sMessage);
		aOutputArgInfo[3].DataType := eUAType_Int16;
		aOutputArgInfo[3].ValueRank := -1;
		aOutputArgInfo[3].nLenData := SIZEOF(stTrafficLightColorData.stOutput.nTrafficLightColor);
		(* Set up output  *)
		MEMSET(ADR(stTrafficLightColorData.stOutput), 0, SIZEOF(stTrafficLightColorData.stOutput));
		stTrafficLightColorData.stOutput.nNumberOfOutputArguments := nNoOfOutputArgs;
		stTrafficLightColorData.stOutput.stOutputArgInfo[1] := aOutputArgInfo[1];
		stTrafficLightColorData.stOutput.stOutputArgInfo[2] := aOutputArgInfo[2];
		stTrafficLightColorData.stOutput.stOutputArgInfo[3] := aOutputArgInfo[3];
	
		(* Execute FB *)
		fbCallMethod.nNumberOfInputArguments := nNoOfInputArgs;
		fbCallMethod.pInputArgInfo := ADR(aInputArgInfo);
		fbCallMethod.cbInputArgInfo := (SIZEOF(aInputArgInfo[1])*nNoOfInputArgs);
		fbCallMethod.pInputArgData := ADR(aInputData);
		fbCallMethod.cbInputArgData := nOffset;
		fbCallMethod.nNumberOfOutputArguments := nNoOfOutputArgs; 
		fbCallMethod.pOutputArgInfo := ADR(aOutputArgInfo); 
		fbCallMethod.cbOutputArgInfo := (SIZEOF(aOutputArgInfo[1]) * nNoOfOutputArgs); 
		fbCallMethod.pOutputArgInfoAndData := ADR(stTrafficLightColorData.stOutput);
		fbCallMethod.cbOutputArgInfoAndData := SIZEOF(stTrafficLightColorData.stOutput);
		
		stTrafficLightColorData.iStatus := 1;
		bCallMethod := TRUE;
		
	ELSIF (stTrafficLightColorData.iStatus = 1) THEN
		// Method call Completed...
		IF (eStateMethod = E_TrackClientState.Connected) THEN
			// Method call OK
			IF (stTrafficLightColorData.stOutput.eStatus = E_MMServerStatus.eMMServerStatus_Success) THEN
				// Method returned OK
				stTrafficLightColorData.iStatus := 2;
			ELSE
				// Method returned with error
				stTrafficLightColorData.iStatus := 3;
				stTrafficLightColorData.stOutput.sMessage;
				stTrafficLightColorData.stOutput.nTrafficLightColor;
			END_IF
		ELSIF (eStateMethod = E_TrackClientState.Error) THEN
			// Method call failed
			stTrafficLightColorData.iStatus := 3;
		END_IF
		
	END_IF
END_IF

M_CallTrafficLightColor := stTrafficLightColorData.iStatus;
END_METHOD

METHOD PROTECTED M_CallUpdateStationBuffer : INT
VAR_INPUT
	sStationID			: STRING(30);
	eBufferType			: E_MMStationBuffer;
	nBufferIndex		: USINT;	
	nVehicleID			: UINT;
	sCarrierID			: STRING(30);
	nTicket				: UINT;
	nPriority			: UINT;
END_VAR
VAR
END_VAR
IF (stUpdateStationBufferData.iStatus = 2) OR (stUpdateStationBufferData.iStatus = 3) THEN
	stUpdateStationBufferData.iStatus := 0;
END_IF

IF (bConnectedMethod AND NOT bBusyMethod) THEN
	IF (stUpdateStationBufferData.iStatus = 0) THEN
	(* Setup method calling parameters *)
		(* Method identifier *)
		sObjectIDentifier := stUpdateStationBufferData.sObjectID;
		sMethodIdentifier := stUpdateStationBufferData.sMethodID;
	
		(* Method Inputs *)
		stUpdateStationBufferData.stInput.sStationID := sStationID;
		stUpdateStationBufferData.stInput.eStationBufferType := eBufferType;
		stUpdateStationBufferData.stInput.nIndex := nBufferIndex;
		stUpdateStationBufferData.stInput.nVehicleID := nVehicleID;
		stUpdateStationBufferData.stInput.sCarrierID := sCarrierID;
		stUpdateStationBufferData.stInput.nTicket := nTicket;
		stUpdateStationBufferData.stInput.nPriority := nPriority;
		
		(* Fill input data area with method arguments *)
		MEMSET(ADR(aInputData), 0 ,SIZEOF(aInputData));
		nOffset := 0;
		nOffset := nOffset + MEMCPY(ADR(aInputData)+nOffset, ADR(stUpdateStationBufferData.stInput),	MIN(SIZEOF(stUpdateStationBufferData.stInput), (SIZEOF(aInputData)-nOffset)) );
		(* Number of input arguments *)
		nNoOfInputArgs := stUpdateStationBufferData.iNoOfInputArgs;
		(* Set up input argument information *)
		MEMSET(ADR(aInputArgInfo), 0, SIZEOF(aInputArgInfo));
		aInputArgInfo[1].DataType := eUAType_String;
		aInputArgInfo[1].ValueRank := -1;	// -1: Scalar 
		aInputArgInfo[1].nLenData := SIZEOF(stUpdateStationBufferData.stInput.sStationID);
		aInputArgInfo[2].DataType := eUAType_UInt16;
		aInputArgInfo[2].ValueRank := -1;	// -1: Scalar 
		aInputArgInfo[2].nLenData := SIZEOF(stUpdateStationBufferData.stInput.eStationBufferType);
		aInputArgInfo[3].DataType := eUAType_Byte;
		aInputArgInfo[3].ValueRank := -1;	// -1: Scalar 
		aInputArgInfo[3].nLenData := SIZEOF(stUpdateStationBufferData.stInput.nIndex);
		aInputArgInfo[4].DataType := eUAType_UInt16;
		aInputArgInfo[4].ValueRank := -1;	// -1: Scalar 
		aInputArgInfo[4].nLenData := SIZEOF(stUpdateStationBufferData.stInput.nVehicleID);
		aInputArgInfo[5].DataType := eUAType_String;
		aInputArgInfo[5].ValueRank := -1;	// -1: Scalar 
		aInputArgInfo[5].nLenData := SIZEOF(stUpdateStationBufferData.stInput.sCarrierID);
		aInputArgInfo[6].DataType := eUAType_UInt16;
		aInputArgInfo[6].ValueRank := -1;	// -1: Scalar 
		aInputArgInfo[6].nLenData := SIZEOF(stUpdateStationBufferData.stInput.nTicket);
		aInputArgInfo[7].DataType := eUAType_UInt16;
		aInputArgInfo[7].ValueRank := -1;	// -1: Scalar 
		aInputArgInfo[7].nLenData := SIZEOF(stUpdateStationBufferData.stInput.nPriority);
		
		(* Method outputs *)
		(* Clear output data area *)
		(* Number of output arguments *)
		nNoOfOutputArgs := stUpdateStationBufferData.iNoOfOutputArgs;
		(* Set up output argument information *)
		MEMSET(ADR(aOutputArgInfo), 0, SIZEOF(aOutputArgInfo));
		aOutputArgInfo[1].DataType := eUAType_Uint16;
		aOutputArgInfo[1].ValueRank := -1;
		aOutputArgInfo[1].nLenData := SIZEOF(stUpdateStationBufferData.stOutput.eStatus);
		aOutputArgInfo[2].DataType := eUAType_String;
		aOutputArgInfo[2].ValueRank := -1;
		aOutputArgInfo[2].nLenData := SIZEOF(stUpdateStationBufferData.stOutput.sMessage);
		(* Set up output  *)
		MEMSET(ADR(stUpdateStationBufferData.stOutput), 0, SIZEOF(stUpdateStationBufferData.stOutput));
		stUpdateStationBufferData.stOutput.nNumberOfOutputArguments := nNoOfOutputArgs;
		stUpdateStationBufferData.stOutput.stOutputArgInfo[1] := aOutputArgInfo[1];
		stUpdateStationBufferData.stOutput.stOutputArgInfo[2] := aOutputArgInfo[2];
	
		(* Execute FB *)
		fbCallMethod.nNumberOfInputArguments := nNoOfInputArgs;
		fbCallMethod.pInputArgInfo := ADR(aInputArgInfo);
		fbCallMethod.cbInputArgInfo := (SIZEOF(aInputArgInfo[1])*nNoOfInputArgs);
		fbCallMethod.pInputArgData := ADR(aInputData);
		fbCallMethod.cbInputArgData := nOffset;
		fbCallMethod.nNumberOfOutputArguments := nNoOfOutputArgs; 
		fbCallMethod.pOutputArgInfo := ADR(aOutputArgInfo); 
		fbCallMethod.cbOutputArgInfo := (SIZEOF(aOutputArgInfo[1]) * nNoOfOutputArgs); 
		fbCallMethod.pOutputArgInfoAndData := ADR(stUpdateStationBufferData.stOutput);
		fbCallMethod.cbOutputArgInfoAndData := SIZEOF(stUpdateStationBufferData.stOutput);
		
		stUpdateStationBufferData.iStatus := 1;
		bCallMethod := TRUE;
		
	ELSIF (stUpdateStationBufferData.iStatus = 1) THEN
		// Method call Completed...
		IF (eStateMethod = E_TrackClientState.Connected) THEN
			// Method call OK
			IF (stUpdateStationBufferData.stOutput.eStatus = E_MMServerStatus.eMMServerStatus_Success) THEN
				// Method returned OK
				stUpdateStationBufferData.iStatus := 2;
			ELSE
				// Method returned with error
				stUpdateStationBufferData.iStatus := 3;
				stUpdateStationBufferData.stOutput.sMessage;
			END_IF
		ELSIF (eStateMethod = E_TrackClientState.Error) THEN
			// Method call failed
			stUpdateStationBufferData.iStatus := 3;
		END_IF
		
	END_IF
ELSE
	M_CallUpdateStationBuffer := -1;
	RETURN;
END_IF

M_CallUpdateStationBuffer := stUpdateStationBufferData.iStatus;
END_METHOD

METHOD M_CallUpdateVehicleMappingData : INT
VAR_INPUT
	nVehicleID			: UINT;										(* Magnemotion Vehicle ID *)
	sCarrierID			: STRING(30);								(* Carrier ID *)
	bTool				: BOOL;										(*  *)
	sToolID				: STRING(30);								(* Tool ID *)
	bMaterial			: BOOL;										(*  *)
	sMaterialID			: STRING(30);								(* Material ID string *)
END_VAR
VAR
END_VAR
IF (stUpdateVehicleMappingDataData.iStatus = 2) OR (stUpdateVehicleMappingDataData.iStatus = 3) THEN
	stUpdateVehicleMappingDataData.iStatus := 0;
END_IF

IF (bConnectedMethod AND NOT bBusyMethod) THEN
	IF (stUpdateVehicleMappingDataData.iStatus = 0) THEN
	(* Setup method calling parameters *)
		(* Method identifier *)
		sObjectIDentifier := stUpdateVehicleMappingDataData.sObjectID;
		sMethodIdentifier := stUpdateVehicleMappingDataData.sMethodID;
	
		(* Method Inputs *)
		stUpdateVehicleMappingDataData.stInput.nVehicleID := nVehicleID;
		stUpdateVehicleMappingDataData.stInput.sCarrierID := sCarrierID;
		stUpdateVehicleMappingDataData.stInput.bTool := bTool;
		stUpdateVehicleMappingDataData.stInput.sToolID := sToolID;
		stUpdateVehicleMappingDataData.stInput.bMaterial := bMaterial;
		stUpdateVehicleMappingDataData.stInput.sMaterialID := sMaterialID;
		
		(* Fill input data area with method arguments *)
		MEMSET(ADR(aInputData), 0 ,SIZEOF(aInputData));
		nOffset := 0;
		nOffset := nOffset + MEMCPY(ADR(aInputData)+nOffset, ADR(stUpdateVehicleMappingDataData.stInput),	MIN(SIZEOF(stUpdateVehicleMappingDataData.stInput), (SIZEOF(aInputData)-nOffset)) );
		(* Number of input arguments *)
		nNoOfInputArgs := stUpdateVehicleMappingDataData.iNoOfInputArgs;
		(* Set up input argument information *)
		MEMSET(ADR(aInputArgInfo), 0, SIZEOF(aInputArgInfo));
		aInputArgInfo[1].DataType := eUAType_UInt16;
		aInputArgInfo[1].ValueRank := -1;	// -1: Scalar 
		aInputArgInfo[1].nLenData := SIZEOF(stUpdateVehicleMappingDataData.stInput.nVehicleID);
		aInputArgInfo[2].DataType := eUAType_String;
		aInputArgInfo[2].ValueRank := -1;	// -1: Scalar 
		aInputArgInfo[2].nLenData := SIZEOF(stUpdateVehicleMappingDataData.stInput.sCarrierID);
		aInputArgInfo[3].DataType := eUAType_Boolean;
		aInputArgInfo[3].ValueRank := -1;	// -1: Scalar 
		aInputArgInfo[3].nLenData := SIZEOF(stUpdateVehicleMappingDataData.stInput.bTool);
		aInputArgInfo[4].DataType := eUAType_String;
		aInputArgInfo[4].ValueRank := -1;	// -1: Scalar 
		aInputArgInfo[4].nLenData := SIZEOF(stUpdateVehicleMappingDataData.stInput.sToolID);
		aInputArgInfo[5].DataType := eUAType_Boolean;
		aInputArgInfo[5].ValueRank := -1;	// -1: Scalar 
		aInputArgInfo[5].nLenData := SIZEOF(stUpdateVehicleMappingDataData.stInput.bMaterial);
		aInputArgInfo[6].DataType := eUAType_String;
		aInputArgInfo[6].ValueRank := -1;	// -1: Scalar 
		aInputArgInfo[6].nLenData := SIZEOF(stUpdateVehicleMappingDataData.stInput.sMaterialID);
		
		(* Method outputs *)
		(* Clear output data area *)
		(* Number of output arguments *)
		nNoOfOutputArgs := stUpdateVehicleMappingDataData.iNoOfOutputArgs;
		(* Set up output argument information *)
		MEMSET(ADR(aOutputArgInfo), 0, SIZEOF(aOutputArgInfo));
		aOutputArgInfo[1].DataType := eUAType_Uint16;
		aOutputArgInfo[1].ValueRank := -1;
		aOutputArgInfo[1].nLenData := SIZEOF(stUpdateVehicleMappingDataData.stOutput.eStatus);
		aOutputArgInfo[2].DataType := eUAType_String;
		aOutputArgInfo[2].ValueRank := -1;
		aOutputArgInfo[2].nLenData := SIZEOF(stUpdateVehicleMappingDataData.stOutput.sMessage);
		(* Set up output  *)
		MEMSET(ADR(stUpdateVehicleMappingDataData.stOutput), 0, SIZEOF(stUpdateVehicleMappingDataData.stOutput));
		stUpdateVehicleMappingDataData.stOutput.nNumberOfOutputArguments := nNoOfOutputArgs;
		stUpdateVehicleMappingDataData.stOutput.stOutputArgInfo[1] := aOutputArgInfo[1];
		stUpdateVehicleMappingDataData.stOutput.stOutputArgInfo[2] := aOutputArgInfo[2];
	
		(* Execute FB *)
		fbCallMethod.nNumberOfInputArguments := nNoOfInputArgs;
		fbCallMethod.pInputArgInfo := ADR(aInputArgInfo);
		fbCallMethod.cbInputArgInfo := (SIZEOF(aInputArgInfo[1])*nNoOfInputArgs);
		fbCallMethod.pInputArgData := ADR(aInputData);
		fbCallMethod.cbInputArgData := nOffset;
		fbCallMethod.nNumberOfOutputArguments := nNoOfOutputArgs; 
		fbCallMethod.pOutputArgInfo := ADR(aOutputArgInfo); 
		fbCallMethod.cbOutputArgInfo := (SIZEOF(aOutputArgInfo[1]) * nNoOfOutputArgs); 
		fbCallMethod.pOutputArgInfoAndData := ADR(stUpdateVehicleMappingDataData.stOutput);
		fbCallMethod.cbOutputArgInfoAndData := SIZEOF(stUpdateVehicleMappingDataData.stOutput);
		
		stUpdateVehicleMappingDataData.iStatus := 1;
		bCallMethod := TRUE;
		
	ELSIF (stUpdateVehicleMappingDataData.iStatus = 1) THEN
		// Method call Completed...
		IF (eStateMethod = E_TrackClientState.Connected) THEN
			// Method call OK
			IF (stUpdateVehicleMappingDataData.stOutput.eStatus = E_MMServerStatus.eMMServerStatus_Success) THEN
				// Method returned OK
				stUpdateVehicleMappingDataData.iStatus := 2;
				// Trig vehicle data reading because data has changed
				M_VehicleToReadAdd(stUpdateVehicleMappingDataData.stInput.nVehicleID);
				
			ELSE
				// Method returned with error
				stUpdateVehicleMappingDataData.iStatus := 3;
				stUpdateVehicleMappingDataData.stOutput.sMessage;
				
			END_IF
			
		ELSIF (eStateMethod = E_TrackClientState.Error) THEN
			// Method call failed
			stUpdateVehicleMappingDataData.iStatus := 3;
			
		END_IF
		
	END_IF
ELSE
	M_CallUpdateVehicleMappingData := -1;
	RETURN;
	
END_IF

M_CallUpdateVehicleMappingData := stUpdateVehicleMappingDataData.iStatus;
END_METHOD

METHOD M_CallUpdateVehicleMontage : INT
VAR_INPUT
	nVehicleID			: UINT;										(* Magnemotion Vehicle ID *)
	bTool				: BOOL;										(*  *)
	sToolID				: STRING(30);								(* Tool ID *)
	bMaterial			: BOOL;										(*  *)
	sMaterialID			: STRING(30);								(* Material ID string *)
	bReserved			: BOOL;										(* TRUE signals vehicle is reserved for montage line *)
END_VAR
VAR
END_VAR
IF (stUpdateVehicleMontageData.iStatus = 2) OR (stUpdateVehicleMontageData.iStatus = 3) THEN
	stUpdateVehicleMontageData.iStatus := 0;
END_IF

IF (bConnectedMethod AND NOT bBusyMethod) THEN
	IF (stUpdateVehicleMontageData.iStatus = 0) THEN
	(* Setup method calling parameters *)
		(* Method identifier *)
		sObjectIDentifier := stUpdateVehicleMontageData.sObjectID;
		sMethodIdentifier := stUpdateVehicleMontageData.sMethodID;
	
		(* Method Inputs *)
		stUpdateVehicleMontageData.stInput.eInputType := E_MMVehicleInputType.eMMVehicleInputType_VehicleID;
		stUpdateVehicleMontageData.stInput.sInput := UINT_TO_STRING(nVehicleID);
		stUpdateVehicleMontageData.stInput.bTool := bTool;
		stUpdateVehicleMontageData.stInput.sToolID := sToolID;
		stUpdateVehicleMontageData.stInput.bMaterial := bMaterial;
		stUpdateVehicleMontageData.stInput.sMaterialID := sMaterialID;
		stUpdateVehicleMontageData.stInput.bReserved := bReserved;
		
		(* Fill input data area with method arguments *)
		MEMSET(ADR(aInputData), 0 ,SIZEOF(aInputData));
		nOffset := 0;
		nOffset := nOffset + MEMCPY(ADR(aInputData)+nOffset, ADR(stUpdateVehicleMontageData.stInput),	MIN(SIZEOF(stUpdateVehicleMontageData.stInput), (SIZEOF(aInputData)-nOffset)) );
		(* Number of input arguments *)
		nNoOfInputArgs := stUpdateVehicleMontageData.iNoOfInputArgs;
		(* Set up input argument information *)
		MEMSET(ADR(aInputArgInfo), 0, SIZEOF(aInputArgInfo));
		aInputArgInfo[1].DataType := eUAType_UInt16;
		aInputArgInfo[1].ValueRank := -1;	// -1: Scalar 
		aInputArgInfo[1].nLenData := SIZEOF(stUpdateVehicleMontageData.stInput.eInputType);
		aInputArgInfo[2].DataType := eUAType_String;
		aInputArgInfo[2].ValueRank := -1;	// -1: Scalar 
		aInputArgInfo[2].nLenData := SIZEOF(stUpdateVehicleMontageData.stInput.sInput);
		aInputArgInfo[3].DataType := eUAType_Boolean;
		aInputArgInfo[3].ValueRank := -1;	// -1: Scalar 
		aInputArgInfo[3].nLenData := SIZEOF(stUpdateVehicleMontageData.stInput.bTool);
		aInputArgInfo[4].DataType := eUAType_String;
		aInputArgInfo[4].ValueRank := -1;	// -1: Scalar 
		aInputArgInfo[4].nLenData := SIZEOF(stUpdateVehicleMontageData.stInput.sToolID);
		aInputArgInfo[5].DataType := eUAType_Boolean;
		aInputArgInfo[5].ValueRank := -1;	// -1: Scalar 
		aInputArgInfo[5].nLenData := SIZEOF(stUpdateVehicleMontageData.stInput.bMaterial);
		aInputArgInfo[6].DataType := eUAType_String;
		aInputArgInfo[6].ValueRank := -1;	// -1: Scalar 
		aInputArgInfo[6].nLenData := SIZEOF(stUpdateVehicleMontageData.stInput.sMaterialID);
		aInputArgInfo[7].DataType := eUAType_Boolean;
		aInputArgInfo[7].ValueRank := -1;	// -1: Scalar 
		aInputArgInfo[7].nLenData := SIZEOF(stUpdateVehicleMontageData.stInput.bReserved);
		
		(* Method outputs *)
		(* Clear output data area *)
		(* Number of output arguments *)
		nNoOfOutputArgs := stUpdateVehicleMontageData.iNoOfOutputArgs;
		(* Set up output argument information *)
		MEMSET(ADR(aOutputArgInfo), 0, SIZEOF(aOutputArgInfo));
		aOutputArgInfo[1].DataType := eUAType_Uint16;
		aOutputArgInfo[1].ValueRank := -1;
		aOutputArgInfo[1].nLenData := SIZEOF(stUpdateVehicleMontageData.stOutput.eStatus);
		aOutputArgInfo[2].DataType := eUAType_String;
		aOutputArgInfo[2].ValueRank := -1;
		aOutputArgInfo[2].nLenData := SIZEOF(stUpdateVehicleMontageData.stOutput.sMessage);
		(* Set up output  *)
		MEMSET(ADR(stUpdateVehicleMontageData.stOutput), 0, SIZEOF(stUpdateVehicleMontageData.stOutput));
		stUpdateVehicleMontageData.stOutput.nNumberOfOutputArguments := nNoOfOutputArgs;
		stUpdateVehicleMontageData.stOutput.stOutputArgInfo[1] := aOutputArgInfo[1];
		stUpdateVehicleMontageData.stOutput.stOutputArgInfo[2] := aOutputArgInfo[2];
	
		(* Execute FB *)
		fbCallMethod.nNumberOfInputArguments := nNoOfInputArgs;
		fbCallMethod.pInputArgInfo := ADR(aInputArgInfo);
		fbCallMethod.cbInputArgInfo := (SIZEOF(aInputArgInfo[1])*nNoOfInputArgs);
		fbCallMethod.pInputArgData := ADR(aInputData);
		fbCallMethod.cbInputArgData := nOffset;
		fbCallMethod.nNumberOfOutputArguments := nNoOfOutputArgs; 
		fbCallMethod.pOutputArgInfo := ADR(aOutputArgInfo); 
		fbCallMethod.cbOutputArgInfo := (SIZEOF(aOutputArgInfo[1]) * nNoOfOutputArgs); 
		fbCallMethod.pOutputArgInfoAndData := ADR(stUpdateVehicleMontageData.stOutput);
		fbCallMethod.cbOutputArgInfoAndData := SIZEOF(stUpdateVehicleMontageData.stOutput);
		
		stUpdateVehicleMontageData.iStatus := 1;
		bCallMethod := TRUE;
		
	ELSIF (stUpdateVehicleMontageData.iStatus = 1) THEN
		// Method call Completed...
		IF (UINT_TO_STRING(nVehicleID) = stUpdateVehicleMontageData.stInput.sInput) THEN
			IF (eStateMethod = E_TrackClientState.Connected) THEN
				// Method call OK
				IF (stUpdateVehicleMontageData.stOutput.eStatus = E_MMServerStatus.eMMServerStatus_Success) THEN
					// Method returned OK
					stUpdateVehicleMontageData.iStatus := 2;
					// Trig vehicle data reading because data has changed
					M_VehicleToReadAdd(nVehicleID);
									
				ELSE
					// Method returned with error
					stUpdateVehicleMontageData.iStatus := 3;
					stUpdateVehicleMontageData.stOutput.sMessage;
					
				END_IF
				
			ELSIF (eStateMethod = E_TrackClientState.Error) THEN
				// Method call failed
				stUpdateVehicleMontageData.iStatus := 3;
	
			END_IF
		ELSE
			// Wrong vehicle ID
			F_LogLine('TC_VMD: Wrong Vehicle ID (%d)', nVehicleID);
			
		END_IF
	END_IF
ELSE
	M_CallUpdateVehicleMontage := -1;
	RETURN;

END_IF

M_CallUpdateVehicleMontage := stUpdateVehicleMontageData.iStatus;
END_METHOD

METHOD PROTECTED M_CallUpdateVehicleOwner : INT
VAR_INPUT
	nVehicleID			: UINT;										(* Magnemotion Vehicle ID *)
	eInputType			: E_MMVehicleInputType;
	sInput				: STRING(30);
	sCellID				: STRING(30);
END_VAR
VAR
END_VAR
IF (stUpdateVehicleOwnerData.iStatus = 2) OR (stUpdateVehicleOwnerData.iStatus = 3) THEN
	stUpdateVehicleOwnerData.iStatus := 0;
END_IF

IF (bConnectedMethod AND NOT bBusyMethod) THEN
	IF (stUpdateVehicleOwnerData.iStatus = 0) THEN
	(* Setup method calling parameters *)
		(* Method identifier *)
		sObjectIDentifier := stUpdateVehicleOwnerData.sObjectID;
		sMethodIdentifier := stUpdateVehicleOwnerData.sMethodID;
	
		(* Method Inputs *)
		stUpdateVehicleOwnerData.stInput.eInputType := eInputType;
		stUpdateVehicleOwnerData.stInput.sInput := sInput;
		stUpdateVehicleOwnerData.stInput.sCellID := sCellID;
		
		(* Fill input data area with method arguments *)
		MEMSET(ADR(aInputData), 0 ,SIZEOF(aInputData));
		nOffset := 0;
		nOffset := nOffset + MEMCPY(ADR(aInputData)+nOffset, ADR(stUpdateVehicleOwnerData.stInput),	MIN(SIZEOF(stUpdateVehicleOwnerData.stInput), (SIZEOF(aInputData)-nOffset)) );
		(* Number of input arguments *)
		nNoOfInputArgs := stUpdateVehicleOwnerData.iNoOfInputArgs;
		(* Set up input argument information *)
		MEMSET(ADR(aInputArgInfo), 0, SIZEOF(aInputArgInfo));
		aInputArgInfo[1].DataType := eUAType_UInt16;
		aInputArgInfo[1].ValueRank := -1;	// -1: Scalar 
		aInputArgInfo[1].nLenData := SIZEOF(stUpdateVehicleOwnerData.stInput.eInputType);
		aInputArgInfo[2].DataType := eUAType_String;
		aInputArgInfo[2].ValueRank := -1;	// -1: Scalar 
		aInputArgInfo[2].nLenData := SIZEOF(stUpdateVehicleOwnerData.stInput.sInput);
		aInputArgInfo[3].DataType := eUAType_String;
		aInputArgInfo[3].ValueRank := -1;	// -1: Scalar 
		aInputArgInfo[3].nLenData := SIZEOF(stUpdateVehicleOwnerData.stInput.sCellID);
		
		(* Method outputs *)
		(* Clear output data area *)
		(* Number of output arguments *)
		nNoOfOutputArgs := stUpdateVehicleOwnerData.iNoOfOutputArgs;
		(* Set up output argument information *)
		MEMSET(ADR(aOutputArgInfo), 0, SIZEOF(aOutputArgInfo));
		aOutputArgInfo[1].DataType := eUAType_Uint16;
		aOutputArgInfo[1].ValueRank := -1;
		aOutputArgInfo[1].nLenData := SIZEOF(stUpdateVehicleOwnerData.stOutput.eStatus);
		aOutputArgInfo[2].DataType := eUAType_String;
		aOutputArgInfo[2].ValueRank := -1;
		aOutputArgInfo[2].nLenData := SIZEOF(stUpdateVehicleOwnerData.stOutput.sMessage);
		(* Set up output  *)
		MEMSET(ADR(stUpdateVehicleOwnerData.stOutput), 0, SIZEOF(stUpdateVehicleOwnerData.stOutput));
		stUpdateVehicleOwnerData.stOutput.nNumberOfOutputArguments := nNoOfOutputArgs;
		stUpdateVehicleOwnerData.stOutput.stOutputArgInfo[1] := aOutputArgInfo[1];
		stUpdateVehicleOwnerData.stOutput.stOutputArgInfo[2] := aOutputArgInfo[2];
	
		(* Execute FB *)
		fbCallMethod.nNumberOfInputArguments := nNoOfInputArgs;
		fbCallMethod.pInputArgInfo := ADR(aInputArgInfo);
		fbCallMethod.cbInputArgInfo := (SIZEOF(aInputArgInfo[1])*nNoOfInputArgs);
		fbCallMethod.pInputArgData := ADR(aInputData);
		fbCallMethod.cbInputArgData := nOffset;
		fbCallMethod.nNumberOfOutputArguments := nNoOfOutputArgs; 
		fbCallMethod.pOutputArgInfo := ADR(aOutputArgInfo); 
		fbCallMethod.cbOutputArgInfo := (SIZEOF(aOutputArgInfo[1]) * nNoOfOutputArgs); 
		fbCallMethod.pOutputArgInfoAndData := ADR(stUpdateVehicleOwnerData.stOutput);
		fbCallMethod.cbOutputArgInfoAndData := SIZEOF(stUpdateVehicleOwnerData.stOutput);
		
		stUpdateVehicleOwnerData.iStatus := 1;
		bCallMethod := TRUE;
		
	ELSIF (stUpdateVehicleOwnerData.iStatus = 1) THEN
		// Method call Completed...
		IF (eStateMethod = E_TrackClientState.Connected) THEN
			// Method call OK
			IF (stUpdateVehicleOwnerData.stOutput.eStatus = E_MMServerStatus.eMMServerStatus_Success) THEN
				// Method returned OK
				stUpdateVehicleOwnerData.iStatus := 2;
				// Trig vehicle data reading because data has changed
				M_VehicleToReadAdd(nVehicleID);
				
			ELSE
				// Method returned with error
				stUpdateVehicleOwnerData.iStatus := 3;
				stUpdateVehicleOwnerData.stOutput.sMessage;

			END_IF
		ELSIF (eStateMethod = E_TrackClientState.Error) THEN
			// Method call failed
			stUpdateVehicleOwnerData.iStatus := 3;

		END_IF
		
	END_IF
ELSE
	M_CallUpdateVehicleOwner := -1;
	RETURN;

END_IF

M_CallUpdateVehicleOwner := stUpdateVehicleOwnerData.iStatus;
END_METHOD

METHOD M_CallUpdateVehicleReservationData : INT
VAR_INPUT
	nVehicleID			: UINT;										(* Magnemotion vehicle ID *)
	sTargetStationID	: STRING(30);								(* Target station ID *)
	sCarrierID			: STRING(30);								(* Carrier ID *)
	sJobID				: STRING(30);								(* Job ID string *)
	nTicket				: UINT;										(* Ticket number *)
	nCarriersInPackage	: UINT;										(* Ticket size *)
	nPriority			: UINT;										(* Ticket priority *)
END_VAR
VAR
END_VAR
IF (stUpdateVehicleReservationDataData.iStatus = 2) OR (stUpdateVehicleReservationDataData.iStatus = 3) THEN
	stUpdateVehicleReservationDataData.iStatus := 0;
END_IF

IF (bConnectedMethod AND NOT bBusyMethod) THEN
	IF (stUpdateVehicleReservationDataData.iStatus = 0) THEN
	(* Setup method calling parameters *)
		(* Method identifier *)
		sObjectIDentifier := stUpdateVehicleReservationDataData.sObjectID;
		sMethodIdentifier := stUpdateVehicleReservationDataData.sMethodID;
	
		(* Method Inputs *)
		stUpdateVehicleReservationDataData.stInput.sTargetStationID := sTargetStationID;
		stUpdateVehicleReservationDataData.stInput.sCarrierID := sCarrierID;
		stUpdateVehicleReservationDataData.stInput.sJobID := sJobID;
		stUpdateVehicleReservationDataData.stInput.nTicket := nTicket;
		stUpdateVehicleReservationDataData.stInput.nCarriersInPackage := nCarriersInPackage;
		stUpdateVehicleReservationDataData.stInput.nPriority := nPriority;
		
		(* Fill input data area with method arguments *)
		MEMSET(ADR(aInputData), 0 ,SIZEOF(aInputData));
		nOffset := 0;
		nOffset := nOffset + MEMCPY(ADR(aInputData)+nOffset, ADR(stUpdateVehicleReservationDataData.stInput),	MIN(SIZEOF(stUpdateVehicleReservationDataData.stInput), (SIZEOF(aInputData)-nOffset)) );
		(* Number of input arguments *)
		nNoOfInputArgs := stUpdateVehicleReservationDataData.iNoOfInputArgs;
		(* Set up input argument information *)
		MEMSET(ADR(aInputArgInfo), 0, SIZEOF(aInputArgInfo));
		aInputArgInfo[1].DataType := eUAType_String;
		aInputArgInfo[1].ValueRank := -1;	// -1: Scalar 
		aInputArgInfo[1].nLenData := SIZEOF(stUpdateVehicleReservationDataData.stInput.sTargetStationID);
		aInputArgInfo[2].DataType := eUAType_String;
		aInputArgInfo[2].ValueRank := -1;	// -1: Scalar 
		aInputArgInfo[2].nLenData := SIZEOF(stUpdateVehicleReservationDataData.stInput.sCarrierID);
		aInputArgInfo[3].DataType := eUAType_String;
		aInputArgInfo[3].ValueRank := -1;	// -1: Scalar 
		aInputArgInfo[3].nLenData := SIZEOF(stUpdateVehicleReservationDataData.stInput.sJobID);
		aInputArgInfo[4].DataType := eUAType_UInt16;
		aInputArgInfo[4].ValueRank := -1;	// -1: Scalar 
		aInputArgInfo[4].nLenData := SIZEOF(stUpdateVehicleReservationDataData.stInput.nTicket);
		aInputArgInfo[5].DataType := eUAType_UInt16;
		aInputArgInfo[5].ValueRank := -1;	// -1: Scalar 
		aInputArgInfo[5].nLenData := SIZEOF(stUpdateVehicleReservationDataData.stInput.nCarriersInPackage);
		aInputArgInfo[6].DataType := eUAType_UInt16;
		aInputArgInfo[6].ValueRank := -1;	// -1: Scalar 
		aInputArgInfo[6].nLenData := SIZEOF(stUpdateVehicleReservationDataData.stInput.nPriority);
		
		(* Method outputs *)
		(* Clear output data area *)
		(* Number of output arguments *)
		nNoOfOutputArgs := stUpdateVehicleReservationDataData.iNoOfOutputArgs;
		(* Set up output argument information *)
		MEMSET(ADR(aOutputArgInfo), 0, SIZEOF(aOutputArgInfo));
		aOutputArgInfo[1].DataType := eUAType_Uint16;
		aOutputArgInfo[1].ValueRank := -1;
		aOutputArgInfo[1].nLenData := SIZEOF(stUpdateVehicleReservationDataData.stOutput.eStatus);
		aOutputArgInfo[2].DataType := eUAType_String;
		aOutputArgInfo[2].ValueRank := -1;
		aOutputArgInfo[2].nLenData := SIZEOF(stUpdateVehicleReservationDataData.stOutput.sMessage);
		(* Set up output  *)
		MEMSET(ADR(stUpdateVehicleReservationDataData.stOutput), 0, SIZEOF(stUpdateVehicleReservationDataData.stOutput));
		stUpdateVehicleReservationDataData.stOutput.nNumberOfOutputArguments := nNoOfOutputArgs;
		stUpdateVehicleReservationDataData.stOutput.stOutputArgInfo[1] := aOutputArgInfo[1];
		stUpdateVehicleReservationDataData.stOutput.stOutputArgInfo[2] := aOutputArgInfo[2];
	
		(* Execute FB *)
		fbCallMethod.nNumberOfInputArguments := nNoOfInputArgs;
		fbCallMethod.pInputArgInfo := ADR(aInputArgInfo);
		fbCallMethod.cbInputArgInfo := (SIZEOF(aInputArgInfo[1])*nNoOfInputArgs);
		fbCallMethod.pInputArgData := ADR(aInputData);
		fbCallMethod.cbInputArgData := nOffset;
		fbCallMethod.nNumberOfOutputArguments := nNoOfOutputArgs; 
		fbCallMethod.pOutputArgInfo := ADR(aOutputArgInfo); 
		fbCallMethod.cbOutputArgInfo := (SIZEOF(aOutputArgInfo[1]) * nNoOfOutputArgs); 
		fbCallMethod.pOutputArgInfoAndData := ADR(stUpdateVehicleReservationDataData.stOutput);
		fbCallMethod.cbOutputArgInfoAndData := SIZEOF(stUpdateVehicleReservationDataData.stOutput);
		
		stUpdateVehicleReservationDataData.iStatus := 1;
		bCallMethod := TRUE;
		
	ELSIF (stUpdateVehicleReservationDataData.iStatus = 1) THEN
		// Method call Completed...
		IF (eStateMethod = E_TrackClientState.Connected) THEN
			// Method call OK
			IF (stUpdateVehicleReservationDataData.stOutput.eStatus = E_MMServerStatus.eMMServerStatus_Success) THEN
				// Method returned OK
				stUpdateVehicleReservationDataData.iStatus := 2;
				// Trig vehicle data reading because data has changed
				M_VehicleToReadAdd(nVehicleID);
				
			ELSE
				// Method returned with error
				stUpdateVehicleReservationDataData.iStatus := 3;
				stUpdateVehicleReservationDataData.stOutput.sMessage;

			END_IF

		ELSIF (eStateMethod = E_TrackClientState.Error) THEN
			// Method call failed
			stUpdateVehicleReservationDataData.iStatus := 3;

		END_IF
		
	END_IF
ELSE
	M_CallUpdateVehicleReservationData := -1;
	RETURN;

END_IF

M_CallUpdateVehicleReservationData := stUpdateVehicleReservationDataData.iStatus;
END_METHOD

METHOD M_CallUpdateVehicleReworkData : INT
VAR_INPUT
	nVehicleID			: UINT;										(* Magnemotion Vehicle ID *)
	sCarrierID			: STRING(30);								(* Carrier ID *)
	bNOK				: BOOL;										(* TRUE signals that rework is required *)
END_VAR
VAR
END_VAR
IF (stUpdateVehicleReworkDataData.iStatus = 2) OR (stUpdateVehicleReworkDataData.iStatus = 3) THEN
	stUpdateVehicleReworkDataData.iStatus := 0;
END_IF

IF (bConnectedMethod AND NOT bBusyMethod) THEN
	IF (stUpdateVehicleReworkDataData.iStatus = 0) THEN
	(* Setup method calling parameters *)
		(* Method identifier *)
		sObjectIDentifier := stUpdateVehicleReworkDataData.sObjectID;
		sMethodIdentifier := stUpdateVehicleReworkDataData.sMethodID;
	
		(* Method Inputs *)
		stUpdateVehicleReworkDataData.stInput.sCarrierID := sCarrierID;
		stUpdateVehicleReworkDataData.stInput.bNOK := bNOK;
		
		(* Fill input data area with method arguments *)
		MEMSET(ADR(aInputData), 0 ,SIZEOF(aInputData));
		nOffset := 0;
		nOffset := nOffset + MEMCPY(ADR(aInputData)+nOffset, ADR(stUpdateVehicleReworkDataData.stInput),	MIN(SIZEOF(stUpdateVehicleReworkDataData.stInput), (SIZEOF(aInputData)-nOffset)) );
		(* Number of input arguments *)
		nNoOfInputArgs := stUpdateVehicleReworkDataData.iNoOfInputArgs;
		(* Set up input argument information *)
		MEMSET(ADR(aInputArgInfo), 0, SIZEOF(aInputArgInfo));
		aInputArgInfo[1].DataType := eUAType_String;
		aInputArgInfo[1].ValueRank := -1;	// -1: Scalar 
		aInputArgInfo[1].nLenData := SIZEOF(stUpdateVehicleReworkDataData.stInput.sCarrierID);
		aInputArgInfo[2].DataType := eUAType_Boolean;
		aInputArgInfo[2].ValueRank := -1;	// -1: Scalar 
		aInputArgInfo[2].nLenData := SIZEOF(stUpdateVehicleReworkDataData.stInput.bNOK);
		
		(* Method outputs *)
		(* Clear output data area *)
		(* Number of output arguments *)
		nNoOfOutputArgs := stUpdateVehicleReworkDataData.iNoOfOutputArgs;
		(* Set up output argument information *)
		MEMSET(ADR(aOutputArgInfo), 0, SIZEOF(aOutputArgInfo));
		aOutputArgInfo[1].DataType := eUAType_Uint16;
		aOutputArgInfo[1].ValueRank := -1;
		aOutputArgInfo[1].nLenData := SIZEOF(stUpdateVehicleReworkDataData.stOutput.eStatus);
		aOutputArgInfo[2].DataType := eUAType_String;
		aOutputArgInfo[2].ValueRank := -1;
		aOutputArgInfo[2].nLenData := SIZEOF(stUpdateVehicleReworkDataData.stOutput.sMessage);
		(* Set up output  *)
		MEMSET(ADR(stUpdateVehicleReworkDataData.stOutput), 0, SIZEOF(stUpdateVehicleReworkDataData.stOutput));
		stUpdateVehicleReworkDataData.stOutput.nNumberOfOutputArguments := nNoOfOutputArgs;
		stUpdateVehicleReworkDataData.stOutput.stOutputArgInfo[1] := aOutputArgInfo[1];
		stUpdateVehicleReworkDataData.stOutput.stOutputArgInfo[2] := aOutputArgInfo[2];
	
		(* Execute FB *)
		fbCallMethod.nNumberOfInputArguments := nNoOfInputArgs;
		fbCallMethod.pInputArgInfo := ADR(aInputArgInfo);
		fbCallMethod.cbInputArgInfo := (SIZEOF(aInputArgInfo[1])*nNoOfInputArgs);
		fbCallMethod.pInputArgData := ADR(aInputData);
		fbCallMethod.cbInputArgData := nOffset;
		fbCallMethod.nNumberOfOutputArguments := nNoOfOutputArgs; 
		fbCallMethod.pOutputArgInfo := ADR(aOutputArgInfo); 
		fbCallMethod.cbOutputArgInfo := (SIZEOF(aOutputArgInfo[1]) * nNoOfOutputArgs); 
		fbCallMethod.pOutputArgInfoAndData := ADR(stUpdateVehicleReworkDataData.stOutput);
		fbCallMethod.cbOutputArgInfoAndData := SIZEOF(stUpdateVehicleReworkDataData.stOutput);
		
		stUpdateVehicleReworkDataData.iStatus := 1;
		bCallMethod := TRUE;
		
	ELSIF (stUpdateVehicleReworkDataData.iStatus = 1) THEN
		// Method call Completed...
		IF (eStateMethod = E_TrackClientState.Connected) THEN
			// Method call OK
			IF (stUpdateVehicleReworkDataData.stOutput.eStatus = E_MMServerStatus.eMMServerStatus_Success) THEN
				// Method returned OK
				stUpdateVehicleReworkDataData.iStatus := 2;
				// Trig vehicle data reading because data has changed
				M_VehicleToReadAdd(nVehicleID);
								
			ELSE
				// Method returned with error
				stUpdateVehicleReworkDataData.iStatus := 3;
				stUpdateVehicleReworkDataData.stOutput.sMessage;
				
			END_IF
			
		ELSIF (eStateMethod = E_TrackClientState.Error) THEN
			// Method call failed
			stUpdateVehicleReworkDataData.iStatus := 3;

		END_IF
		
	END_IF
ELSE
	M_CallUpdateVehicleReworkData := -1;
	RETURN;

END_IF

M_CallUpdateVehicleReworkData := stUpdateVehicleReworkDataData.iStatus;
END_METHOD

METHOD PROTECTED M_CarrierIDToVehicleID : UINT
VAR_INPUT
	sCarrierID		: STRING(30);
END_VAR

VAR
	i: INT;
END_VAR

// Find vehicle with specified Carrier ID
FOR i := 1 TO MM_MAX_NUMBER_OF_VEHICLE_ELEMENTS BY 1 DO
	IF (aReadVehicleData[i].stVehicle.bDataValid) THEN
		IF (F_StringCompNoCase(aReadVehicleData[i].stVehicle.sCarrierID, sCarrierID) ) THEN
			M_CarrierIDToVehicleID := aReadVehicleData[i].stVehicle.nVehicleID;
			RETURN;
		END_IF
	END_IF
END_FOR

// Not found!
M_CarrierIDToVehicleID := 0;
END_METHOD

/// Check if a specified station index belongs to this cell
METHOD PROTECTED M_CheckStationIndex : BOOL
VAR_INPUT
	iStationNo		: UINT;
END_VAR
VAR
	i				: UINT;
END_VAR

FOR i := 1 TO 5 BY 1 DO
	IF (aStations[i].bPresent) THEN
		IF (iThisStationIndex[i] = iStationNo) THEN
			// Station index found
			M_CheckStationIndex := TRUE;
			RETURN;			
		END_IF
	END_IF
END_FOR

// Not found
M_CheckStationIndex := FALSE;
RETURN;
END_METHOD

/// Check if indexes are found for all specified stations
METHOD PROTECTED M_CheckStationsRead : BOOL
VAR
	i				: UINT;
	bReturn			: BOOL;
END_VAR

bReturn := TRUE;

FOR i := 1 TO 5 BY 1 DO
	IF (aStations[i].bPresent) THEN
		IF (iThisStationIndex[i] > 0) THEN
			// Station index found
		ELSE
			// Index for this station is not found!
			bReturn := FALSE;
			EXIT;
		END_IF
	END_IF
END_FOR

// Not found
M_CheckStationsRead := bReturn;
RETURN;
END_METHOD

/// Check if specified vehicle is Owned by this cell and is to be read (evet-driven reading)
METHOD PROTECTED M_CheckVehicleEventRead : BOOL
VAR_INPUT
	iVehicleNo		: UINT;		// MagneMotion Vehicle number
END_VAR
VAR
	i				: UINT;
	bVehicleOwned	: BOOL;
	bVehicleDoRead	: BOOL;
END_VAR

FOR i := 1 TO MM_MAX_NUMBER_OF_VEHICLE_ELEMENTS BY 1 DO
	IF (anVehiclesToRead[i] = iVehicleNo) THEN
		// Vehicle is found in to-read list
		M_CheckVehicleEventRead := TRUE;
		RETURN;
	END_IF

END_FOR

// Not found
M_CheckVehicleEventRead := FALSE;
RETURN;
END_METHOD

/// Check if specified vehicle is Owned by this cell
METHOD PROTECTED M_CheckVehicleOwned : BOOL
VAR_INPUT
	iVehicleNo		: UINT;		// MagneMotion Vehicle number
END_VAR
VAR
	i				: UINT;
END_VAR

FOR i := 1 TO MM_MAX_NUMBER_OF_VEHICLE_ELEMENTS BY 1 DO
	IF (aReadCellData.stCell.anVehicles[i] = iVehicleNo) THEN
		// Vehicle is found
		M_CheckVehicleOwned := TRUE;
		RETURN;
	END_IF
END_FOR

// Not found
M_CheckVehicleOwned := FALSE;
RETURN;
END_METHOD

/// Check if specified vehicle is survailed by this cell
METHOD PROTECTED M_CheckVehicleSurvail : BOOL
VAR_INPUT
	iVehicleNo		: UINT;		// MagneMotion Vehicle number
END_VAR
VAR
	i				: UINT;
END_VAR

FOR i := 1 TO MM_MAX_NUMBER_OF_VEHICLE_ELEMENTS BY 1 DO
	IF (anExtraVehicles[i] = iVehicleNo) THEN
		// Vehicle is found
		M_CheckVehicleSurvail := TRUE;
		RETURN;
	END_IF
END_FOR

// Not found
M_CheckVehicleSurvail := FALSE;
RETURN;
END_METHOD

METHOD M_ClearAll : BOOL
VAR_INPUT
END_VAR
VAR
	i	: UINT;
END_VAR

//Clear data on station(s)
FOR i:=1 TO 5 DO
	IF aStations[i].bPresent THEN
		// Station data
		aStations[i].stStationData1.nTicket := 0;
		aStations[i].stStationData1.nTicketSize := 0;
		aStations[i].stStationData1.CurrentPriority := 0;
		aStations[i].stStationData1.nCurrentVehicleID := 0;
		aStations[i].stStationData1.nReservedVehicleID := 0;
		aStations[i].stStationData2.nTicket := 0;
		aStations[i].stStationData2.nTicketSize := 0;
		aStations[i].stStationData2.CurrentPriority := 0;
		aStations[i].stStationData2.nCurrentVehicleID := 0;
		aStations[i].stStationData2.nReservedVehicleID := 0;
		
		// Station in/output
		bReadyStationIn[i] := FALSE;
		bReadyStationOut[i] := FALSE;

	END_IF
END_FOR

M_ClearAll := TRUE;
END_METHOD

METHOD PROTECTED M_CommandData
VAR_INPUT
END_VAR
VAR
	i			: USINT;
	iRes		: UINT;
END_VAR
// Handle the command data from OPC UA (stCommand)

CASE eCommandDataState OF
	// Init state
	E_CommandDataState.Undefined:
		eCommandDataState := E_CommandDataState.CheckRequest;		

	// Check command data request
	E_CommandDataState.CheckRequest:
		IF ((stCommand.ChangeRequest <> stStatus.ChangeStatus) AND (stCommand.ChangeRequest > 0)) THEN
			// Check if changes is allowed on mapping data (from LC)
			IF (stAdditionalDataIn.MESHandShakes.DataChangeStatusTransportStatus = stStatus.DataChange) THEN
// NOTE: Changed to match new LC software!!! - Hack!				
//				stStatus.ChangeAcknowledge := stCommand.ChangeRequest;
//				stStatus.DataChange := stStatus.DataChange + 1;
			
				// Find vehicle ID for specified Carrier ID
				iCommandDataVehicleID := M_CarrierIDToVehicleID(stCommand.CarrierID);
				IF ((iCommandDataVehicleID > 0) AND (iCommandDataVehicleID <= MM_MAX_NUMBER_OF_VEHICLE_ELEMENTS)) THEN
					// Specified vehicle found
					IF (F_StringCompNoCase(aReadVehicleData[iCommandDataVehicleID].stVehicle.sOwnerCell, sCellID)) THEN
						// Vehicle belongs to this cell
						stStatus.ValidRequest := TRUE;
						IF (stCommand.Ticket <= 0) THEN
							// Clear reservation data for this carrier (do not add reservation)
							eCommandDataState := E_CommandDataState.UpdateJobData;
						ELSE
							// Add reservation to track server
							eCommandDataState := E_CommandDataState.AddReservation;
						END_IF
					ELSE
						eCommandDataState := E_CommandDataState.Error;
					END_IF
				ELSE
					eCommandDataState := E_CommandDataState.Error;
				END_IF
			END_IF
		END_IF
		
	E_CommandDataState.AddReservation:
		iRes := M_CallAddReservation(	sStationID := stCommand.TargetStation,
										sCarrierID := stCommand.CarrierID,
										nTicket := stCommand.Ticket,
										nTicketSize := stCommand.CarriersInPackage,
										nPriority := stCommand.Priority 	);
		IF (iRes = 2) THEN
			// Success
			eCommandDataState := E_CommandDataState.UpdateJobData;
		ELSIF (iRes = 3) THEN
			// Error!
			F_LogLine('ERROR: AddReservation (Ticket: %d)', stCommand.Ticket);
			eCommandDataState := E_CommandDataState.Error;
		END_IF
	
	E_CommandDataState.UpdateJobData:
		iRes := M_CallUpdateVehicleReservationData(	nVehicleID := iCommandDataVehicleID,
													sTargetStationID := stCommand.TargetStation,
													sCarrierID := stCommand.CarrierID,
													nTicket := stCommand.Ticket,
													nCarriersInPackage := stCommand.CarriersInPackage,
													nPriority := stCommand.Priority,
													sJobID := stCommand.JobID 	);
		IF (iRes = 2) THEN
			// Success
			eCommandDataState := E_CommandDataState.Done;
		ELSIF (iRes = 3) THEN
			// Error!
			F_LogLine('ERROR: UpdateJobData (Ticket: %d)', stCommand.Ticket);
			eCommandDataState := E_CommandDataState.Error;
		END_IF
	
	E_CommandDataState.Done:
		stStatus.LatestTicket := stCommand.Ticket;
		stStatus.NumberOfCarriers := stCommand.CarriersInPackage;
		stStatus.ChangeStatus := stCommand.ChangeRequest;
// NOTE: Changed to match new LC software!!! - Hack!				
		stStatus.ChangeAcknowledge := stCommand.ChangeRequest;
		stStatus.DataChange := stStatus.DataChange + 1;
		eCommandDataState := E_CommandDataState.Undefined;
		
	E_CommandDataState.Error:
		stStatus.ValidRequest := FALSE;
		stStatus.ChangeStatus := stCommand.ChangeRequest;
// NOTE: Changed to match new LC software!!! - Hack!				
		stStatus.ChangeAcknowledge := stCommand.ChangeRequest;
		stStatus.DataChange := stStatus.DataChange + 1;
		eCommandDataState := E_CommandDataState.Undefined;
		
END_CASE
END_METHOD

/// Copy vehicle and ticket information from Source to Target and DELETES information on Source!!
METHOD PROTECTED M_CopyAndClearBufferData : BOOL
VAR_IN_OUT
	stSource		: ST_MMBuffer;
	stTarget		: ST_MMBuffer;
END_VAR

	// Update data for target location
	stTarget.nTicket := stSource.nTicket;
	stTarget.nTicketSize := stSource.nTicketSize;
	stTarget.CurrentPriority := stSource.CurrentPriority;
	stTarget.nReservedVehicleID := stSource.nReservedVehicleID;
	stTarget.nCurrentVehicleID := stSource.nCurrentVehicleID;
	// Clear data for source location
	stSource.nTicket := 0;
	stSource.nTicketSize := 0;
	stSource.CurrentPriority := 0;
	stSource.nCurrentVehicleID := 0;
	stSource.nReservedVehicleID := 0;
END_METHOD

/// Copy vehicle and ticket information from Source to Target and DELETES information on Source!!
METHOD PROTECTED M_CopyBufferData : BOOL
VAR_IN_OUT
	stSource		: ST_MMBuffer;
	stTarget		: ST_MMBuffer;
END_VAR

	// Update data for target location
	stTarget.nTicket := stSource.nTicket;
	stTarget.nTicketSize := stSource.nTicketSize;
	stTarget.CurrentPriority := stSource.CurrentPriority;
	stTarget.nReservedVehicleID := stSource.nReservedVehicleID;
	stTarget.nCurrentVehicleID := stSource.nCurrentVehicleID;
END_METHOD

// Set path to control from this cell
METHOD PUBLIC M_DefinePath : BOOL
VAR_INPUT
	nPathNo				: UINT;		// Path number
END_VAR
VAR
	i					: UINT;
	bFound				: BOOL;
END_VAR

bFound := FALSE;

IF ( (nPathNo > 0) AND (nPathNo <= MM_MAX_NUMBER_OF_PATH_ELEMENTS) ) THEN
	FOR i := 1 TO MM_MAX_NUMBER_OF_PATH_ELEMENTS BY 1 DO
		IF (aPaths[i] = nPathNo) THEN
			// Same path found
			IF (bFound) THEN
				// Already added to list, but found again, delete old value
				aPaths[i] := 0;
			END_IF
			bFound := TRUE;
		ELSIF ( (aPaths[i] = 0) AND NOT bFound ) THEN
			// Free spot found, assign value
			aPaths[i] := nPathNo;
			bFound := TRUE;
		END_IF
	END_FOR
END_IF

M_DefinePath := bFound;
END_METHOD

METHOD PUBLIC M_DefinePathSegment : BOOL
VAR_INPUT
	nPathSegmentNo	: UINT;
	nPathID			: UINT;		// Path number
	rPositionBegin	: REAL;		// Distance on the specified path to begin segment
	rPositionEnd	: REAL;		// Distance on the specified path to end segment
END_VAR
// Check if data is valid
IF ( (nPathID > 0) AND (rPositionBegin >= 0.0) AND (rPositionEnd > rPositionBegin) ) THEN
	IF (nPathSegmentNo = 1) THEN
		stExitPointSeg1LocBegin.nPathID := nPathID;
		stExitPointSeg1LocBegin.fPosition := rPositionBegin;
		stExitPointSeg1LocEnd.nPathID := nPathID;
		stExitPointSeg1LocEnd.fPosition := rPositionEnd;
		M_DefinePathSegment := TRUE;
		
	ELSIF (nPathSegmentNo = 2) THEN
		stExitPointSeg2LocBegin.nPathID := nPathID;
		stExitPointSeg2LocBegin.fPosition := rPositionBegin;
		stExitPointSeg2LocEnd.nPathID := nPathID;
		stExitPointSeg2LocEnd.fPosition := rPositionEnd;
		M_DefinePathSegment := TRUE;
		
	ELSE
		M_DefinePathSegment := FALSE;
		
	END_IF

ELSE
	M_DefinePathSegment := FALSE;
	
END_IF
END_METHOD

// Set data for traffic light
METHOD PUBLIC M_DefineStation : BOOL
VAR_INPUT
	nStationNo			: UINT(1..5);
	sStationID			: STRING(30);
	nLoc1PathID			: UINT;		// Path number for input location
	rLoc1Position		: REAL;		// Distance on the specified path for input location
	nLoc2PathID			: UINT;		// Path number for output location (0 if single station)
	rLoc2Position		: REAL;		// Distance on the specified path for output location (0.0 if single station)
	nLocDecPathID		: UINT;		// Path number for decision point location
	rLocDecPosition		: REAL;		// Distance on the specified path for decision point location
	nPreBufferSize		: UINT;		// Size of pre buffer (number of positions)
	nPostBufferSize		: UINT;		// Size of post buffer (number of positions)
END_VAR
VAR
	i					: UINT;
	bReInit				: BOOL;
END_VAR
IF ( (nLoc1PathID > 0) AND (rLoc1Position >= 0.0) AND
//	 (nLoc2PathID > 0) AND (rLoc2Position >= 0.0) AND	// Allow single position stations!
	 (nLocDecPathID > 0) AND (rLocDecPosition >= 0.0) AND 
	 (nStationNo >= 1) AND (nStationNo <= 5) AND
	 (sStationID <> '') ) THEN
	
	IF ( (aStations[nStationNo].sStationID <> sStationID) OR
		 (aStations[nStationNo].stStationData1.stLocation.nPathID <> nLoc1PathID) OR
		 (aStations[nStationNo].stStationData1.stLocation.fPosition <> rLoc1Position) OR
		 (aStations[nStationNo].stStationData2.stLocation.nPathID <> nLoc2PathID) OR
		 (aStations[nStationNo].stStationData2.stLocation.fPosition <> rLoc2Position) OR
		 (aStations[nStationNo].stDecisionLocation.nPathID <> nLocDecPathID) OR
		 (aStations[nStationNo].stDecisionLocation.fPosition <> rLocDecPosition) OR
		 (aStations[nStationNo].bPresent = FALSE) ) THEN
		
		bReInit := TRUE;
	END_IF

	aStations[nStationNo].sStationID := sStationID;
	aStations[nStationNo].stStationData1.stLocation.nPathID := nLoc1PathID;
	aStations[nStationNo].stStationData1.stLocation.fPosition := rLoc1Position;
	IF (nLoc1PathID > 0) THEN
		aStations[nStationNo].stStationData1.bPresent := TRUE;
	ELSE
		aStations[nStationNo].stStationData1.bPresent := FALSE;		
	END_IF
	aStations[nStationNo].stStationData2.stLocation.nPathID := nLoc2PathID;
	aStations[nStationNo].stStationData2.stLocation.fPosition := rLoc2Position;
	IF (nLoc2PathID > 0) THEN
		aStations[nStationNo].stStationData2.bPresent := TRUE;
	ELSE
		aStations[nStationNo].stStationData2.bPresent := FALSE;		
	END_IF
	aStations[nStationNo].stDecisionLocation.nPathID := nLocDecPathID;
	aStations[nStationNo].stDecisionLocation.fPosition := rLocDecPosition;

	// Buffers	
	FOR i := 1 TO MM_MAX_BUFFER_INDEX BY 1 DO
		IF ( (aStations[nStationNo].astPreBuffer[i].bPresent <> (i <= nPreBufferSize)) OR
			 (aStations[nStationNo].astPostBuffer[i].bPresent <> (i <= nPostBufferSize)) ) THEN
			bReInit := TRUE;
		END_IF
		aStations[nStationNo].astPreBuffer[i].bPresent := (i <= nPreBufferSize);
		aStations[nStationNo].astPostBuffer[i].bPresent := (i <= nPostBufferSize);
	END_FOR
	aStations[nStationNo].bPresent := TRUE;
	
	M_DefineStation := TRUE;
ELSE
	M_DefineStation := FALSE;
END_IF
END_METHOD

// Set data for traffic light
METHOD PUBLIC M_DefineStationBufferAdjust : BOOL
VAR_INPUT
	nStationNo			: UINT(1..5);
	rPreBufferAdjust	: REAL;		// Distance to adjust pre-buffer position (M) - Should be negative for pre-buffer
	rPostBufferAdjust	: REAL;		// Distance to adjust post-buffer position (M) - Should be negative for pre-buffer
END_VAR
VAR
END_VAR
IF ( (nStationNo > 0) AND (nStationNo <= 5) ) THEN
	IF (aStations[nStationNo].bPresent) THEN
		// Station defined
		aStationPreBufAdj[nStationNo] := rPreBufferAdjust;
		aStationPostBufAdj[nStationNo] := rPostBufferAdjust;
		M_DefineStationBufferAdjust := TRUE;
	ELSE
		// Station not defined
		M_DefineStationBufferAdjust := FALSE;
	END_IF
ELSE
	// Outside range
	M_DefineStationBufferAdjust := FALSE;
END_IF
END_METHOD

// Set data for traffic light
METHOD PUBLIC M_DefineTrafficLight : BOOL
VAR_INPUT
	nTrafficLightNo	: UINT;
	nPathID			: UINT;		// Path number
	rPosition		: REAL;		// Distance on the specified path
END_VAR

IF ((nTrafficLightNo > 0) AND (nPathID > 0) AND (rPosition >= 0.0)) THEN
	IF (nTrafficLightNo = 1) THEN
		stTrafficLightLocation.nPathID := nPathID;
		stTrafficLightLocation.fPosition := rPosition;
		M_DefineTrafficLight := TRUE;

	ELSIF (nTrafficLightNo = 2) THEN
		stTrafficLight2Location.nPathID := nPathID;
		stTrafficLight2Location.fPosition := rPosition;
		M_DefineTrafficLight := TRUE;

	ELSE
		M_DefineTrafficLight := FALSE;
		
	END_IF
ELSE
	M_DefineTrafficLight := FALSE;
	
END_IF
END_METHOD

// Set data for enable/disable station
METHOD PUBLIC M_EnableStation : BOOL
VAR_INPUT
	nStationNo			: UINT(1..5);
	bPresent			: BOOL;
END_VAR
VAR
	i					: UINT;
END_VAR
IF (nStationNo <= 5) THEN
	aStations[nStationNo].bPresent := bPresent;
	
	M_EnableStation := TRUE;
ELSE
	M_EnableStation := FALSE;
END_IF
END_METHOD

METHOD PROTECTED M_ErrorWarning
VAR_INPUT
END_VAR
VAR
	bDataChange:BOOL;
END_VAR

bDataChange S= 
M_ErrorWarningObj(arErrorWaringData:= stErrorWarning.ErrorWarningData,
	bActive:= eTrackState = E_TrackState.Error, 
	iErrorWarningType:= 2, 
	diErrorWarningID:= E_AlarmCategory.TrackClient + 0, 
	sDeviceID:= 'Track Client',
	iSeverity:= 2, 
	iNativeID:= 0, 
	sNativeMessage:= 'Error State Machine');
	
bDataChange S= 
M_ErrorWarningObj(arErrorWaringData:= stErrorWarning.ErrorWarningData,
	bActive:= eStateMethod = E_TrackState.Error, 
	iErrorWarningType:= 2, 
	diErrorWarningID:= E_AlarmCategory.TrackClient + 1, 
	sDeviceID:= 'Track Client',
	iSeverity:= 2, 
	iNativeID:= 0, 
	sNativeMessage:= 'Error State Machine Method');
	
bDataChange S= 
M_ErrorWarningObj(arErrorWaringData:= stErrorWarning.ErrorWarningData,
	bActive:= eStateNode = E_TrackState.Error, 
	iErrorWarningType:= 2, 
	diErrorWarningID:= E_AlarmCategory.TrackClient + 2, 
	sDeviceID:= 'Track Client',
	iSeverity:= 2, 
	iNativeID:= 0, 
	sNativeMessage:= 'Error State Machine Node ADS');


stErrorWarning.DataChange := stErrorWarning.DataChange + TO_UINT(bDataChange);
bDataChange := FALSE;
END_METHOD

METHOD M_ErrorWarningObj : BOOL
VAR_INPUT
	bActive				: BOOL;
	iErrorWarningType	: UINT;
	diErrorWarningID 	: UDINT;
	sDeviceID			: STRING(30);
	iSeverity			: UINT;
	iNativeID			: UDINT;
	sNativeMessage		: STRING(80);
END_VAR
VAR_IN_OUT
	arErrorWaringData	: ARRAY [1..255] OF ST_ErrorWarningDataX;
END_VAR
VAR
	iFoundPos			: UINT;
	i					: UINT;
	j					: UINT;
END_VAR
//Look through array to find existing record(s)
FOR i := 1 TO 255 DO
	IF arErrorWaringData[i].ErrorWarningID = 0 THEN
		EXIT;
	END_IF
	//Existing alarm - first
	IF arErrorWaringData[i].ErrorWarningID = diErrorWarningID AND iFoundPos = 0 THEN
		iFoundPos := i;
	//Multiple records - delete
	ELSIF arErrorWaringData[i].ErrorWarningID = diErrorWarningID AND iFoundPos <> 0 THEN
		MEMSET(ADR(arErrorWaringData[i]), 0, SIZEOF(arErrorWaringData[i]));
		M_ErrorWarningObj := TRUE;
	END_IF
END_FOR

//Alarm high
IF bActive THEN
	//New alarm
	IF iFoundPos = 0 THEN
		arErrorWaringData[i].ErrorWarningType := iErrorWarningType;
		arErrorWaringData[i].DeviceID := sDeviceID;
		arErrorWaringData[i].Severity := iSeverity;
		arErrorWaringData[i].NativeID := iNativeID;
		arErrorWaringData[i].NativeMessage := sNativeMessage;
		arErrorWaringData[i].ErrorWarningID := diErrorWarningID;
		arErrorWaringData[i].DateTime := SYSTEMTIME_TO_STRING(fbGetTime.TIMESTR);
		M_ErrorWarningObj := TRUE;
	END_IF
	
//Alarm low
ELSIF NOT bActive AND iFoundPos <> 0 THEN
	MEMSET(ADR(arErrorWaringData[iFoundPos]), 0, SIZEOF(arErrorWaringData[iFoundPos]));
	M_ErrorWarningObj := TRUE;
END_IF

//Defrag
IF M_ErrorWarningObj THEN
	FOR i:= 1 TO 254 DO
		//Find first empty spot
		IF arErrorWaringData[i].ErrorWarningID = 0 THEN
			//Find first record
			FOR j:= i TO 255 DO
				IF arErrorWaringData[j].ErrorWarningID <> 0 THEN
					//Move to empty spot
					arErrorWaringData[i] := arErrorWaringData[j];
					MEMSET(ADR(arErrorWaringData[j]), 0, SIZEOF(arErrorWaringData[j]));
					EXIT;
				END_IF
			END_FOR
		END_IF
		//No more records
		IF j >= 255 THEN
			RETURN;
		END_IF
	END_FOR
END_IF
END_METHOD

/// Add vehicle to be survailed
METHOD PROTECTED M_ExtraVehicleAdd : BOOL
VAR_INPUT
	iVehicleNo		: UINT;
END_VAR
VAR
	i				: UINT;
	bAdded			: BOOL;
	bRemoved		: BOOL;
END_VAR

FOR i := 1 TO MM_MAX_NUMBER_OF_VEHICLE_ELEMENTS BY 1 DO
	// Check if already excists in list
	IF (anExtraVehicles[i] = iVehicleNo) THEN
		anExtraVehicles[i] := 0;
		bRemoved := TRUE;
	END_IF
	// Add to list
	IF ( (NOT bAdded) AND (anExtraVehicles[i] = 0) ) THEN
		anExtraVehicles[i] := iVehicleNo;
		bAdded := TRUE;
	END_IF
	// Check if finished
	IF (bAdded AND bRemoved) THEN
		M_ExtraVehicleAdd := TRUE;
		RETURN;
	END_IF
	
END_FOR

IF (bAdded) THEN
	// Added
	M_ExtraVehicleAdd := TRUE;
	RETURN;
ELSE
	// NOT Added (list is maybe full!)
	M_ExtraVehicleAdd := FALSE;
	RETURN;	
END_IF
END_METHOD

/// Remove vehicle from surveillance list
METHOD PROTECTED M_ExtraVehicleRemove : BOOL
VAR_INPUT
	iVehicleNo		: UINT;
END_VAR
VAR
	i				: UINT;
END_VAR

FOR i := 1 TO MM_MAX_NUMBER_OF_VEHICLE_ELEMENTS BY 1 DO
	IF (anExtraVehicles[i] = iVehicleNo) THEN
		anExtraVehicles[i] := 0;
		M_ExtraVehicleRemove := TRUE;
		RETURN;
	END_IF
END_FOR

// Not found
M_ExtraVehicleRemove := FALSE;
RETURN;
END_METHOD

METHOD PROTECTED M_Init : BOOL
VAR_INPUT
END_VAR
VAR
	i : UINT;
	sTemp : STRING;
END_VAR
IF (NOT bInitDone) THEN
// Client information to stations
	FOR i := 1 TO 5 BY 1 DO
		aStations[i].sCellID := sCellID;
	END_FOR

// OPC UA Method calling information
	(* Use no encryption *)
	stConnectInfoMethod.eSecurityMode 			:= eUASecurityMsgMode_None;
	(*  *)
	stConnectInfoMethod.eSecurityPolicyUri		:= eUASecurityPolicy_None;
	(* USe TCP transport profile *)
	stConnectInfoMethod.eTransportProfileUri	:= eUATransportProfileUri_UATcp;
	(* Application name *)
	stConnectInfoMethod.sApplicationName		:= '';
	(* Connection timeout *)
	stConnectInfoMethod.tConnectTimeout			:= T#1M;
	(* Session timeout *)
	stConnectInfoMethod.tSessionTimeout			:= T#10M;
	(* Method node ID *)
	stObjectNodeID.eIdentifierType				:= E_UAIdentifierType.eUAIdentifierType_String;
	stMethodNodeID.eIdentifierType				:= E_UAIdentifierType.eUAIdentifierType_String;
	(* Method data *)
	M_InitMethodData();
	
// OPC UA Node reading information
	(* Use no encryption *)
	stConnectInfoNodes.eSecurityMode 			:= eUASecurityMsgMode_None;
	(*  *)
	stConnectInfoNodes.eSecurityPolicyUri		:= eUASecurityPolicy_None;
	(* USe TCP transport profile *)
	stConnectInfoNodes.eTransportProfileUri		:= eUATransportProfileUri_UATcp;
	(* Application name *)
	stConnectInfoNodes.sApplicationName			:= '';
	(* Connection timeout *)
	stConnectInfoNodes.tConnectTimeout			:= T#1M;
	(* Session timeout *)
	stConnectInfoNodes.tSessionTimeout			:= T#10M;

	
	bInitDone := TRUE;
END_IF
END_METHOD

METHOD PROTECTED M_InitMethodData : BOOL

(* Method data *)
stAddStationDoubleData.iStatus				:= 0;
stAddStationSingleData.iStatus				:= 0;
stEnableStationData.iStatus					:= 0;
stRemoveStationData.iStatus					:= 0;

stGetCellIndexData.iStatus					:= 0;

stAddPathData.iStatus						:= 0;
stRemovePathData.iStatus					:= 0;
stStartPathData.iStatus						:= 0;
stResetPathData.iStatus						:= 0;
stSuspendPathData.iStatus					:= 0;
stResumePathData.iStatus					:= 0;

stAddTrafficLightData.iStatus				:= 0;
stRemoveTrafficLightData.iStatus			:= 0;
stTrafficLightColorData.iStatus				:= 0;
stSetTrafficLightColorData.iStatus			:= 0;

stMoveToStationInData.iStatus				:= 0;
stMoveToStationOutData.iStatus				:= 0;
stMoveToPositionData.iStatus				:= 0;
stMoveToBufferData.iStatus					:= 0;
stMoveToDecisionPointData.iStatus			:= 0;
stMoveToScannerData.iStatus					:= 0;

//stUpdateVehicleDataData.iStatus			:= 0;
stUpdateVehicleReservationDataData.iStatus	:= 0;
stUpdateVehicleMappingDataData.iStatus		:= 0;
stUpdateVehicleReworkDataData.iStatus		:= 0;
END_METHOD

METHOD PROTECTED M_InitNodeData : BOOL
VAR
	i				: UINT;
	sPrefix 		: STRING;
	
	bReturn			: BOOL;
END_VAR

(* Node data, init to use string identifier and set namespace index *)
FOR i:=1 TO nMaxNodeIDsInList BY 1 DO
	aNodeIDs[i].eIdentifierType := eUAIdentifierType_String;
	aNodeIDs[i].nNamespaceIndex := nNameSpaceIndexNodes;
END_FOR

nNoOfNodes := 0;
cbDataTotal := 0;

// TEST
//eReadType := E_OPC_NodeType.Nodes;
//iReadIndex := 1;

// Comm type selection
CASE eReadType OF
	E_OPC_NodeType.Vehicles:
		// Select vehicle to read data from
		REPEAT
			iReadIndex := iReadIndex+1;
			IF (iReadIndex > MM_MAX_NUMBER_OF_VEHICLE_ELEMENTS) THEN
				EXIT;
			END_IF
			UNTIL (aReadCellData.stCell.anVehicles[iReadIndex] > 0)
		END_REPEAT
		IF (iReadIndex <= MM_MAX_NUMBER_OF_VEHICLE_ELEMENTS) THEN
			// Build remote symbol name
			sPrefix := CONCAT(sObjectIDentifier, '.stTrackStatus');
			// Data pointer for received data
			pReadNodeData := ADR(aReadVehicleData[iReadIndex]);
			// Header data size
			cbDataTotal := SIZEOF(aReadVehicleData[iReadIndex].stReadListReturnInfo);
			
			// Specify nodes to read by variable name
			nNoOfNodes := nNoOfNodes + 1;
			aNodeIDs[nNoOfNodes].sIdentifier := CONCAT(sPrefix, '.aVehicles[');
			aNodeIDs[nNoOfNodes].sIdentifier := CONCAT(aNodeIDs[nNoOfNodes].sIdentifier, UINT_TO_STRING(aReadCellData.stCell.anVehicles[iReadIndex]));
			aNodeIDs[nNoOfNodes].sIdentifier := CONCAT(aNodeIDs[nNoOfNodes].sIdentifier, ']');
			acbDatas[nNoOfNodes] := SIZEOF(aReadVehicleData[iReadIndex]);
			cbDataTotal := cbDataTotal + acbDatas[nNoOfNodes];
			bReturn := TRUE;
		ELSE
			// Read next type
			iReadIndex := 0;
			eReadType := E_OPC_NodeType.Paths;
			bReturn := FALSE;
		END_IF			
		
	E_OPC_NodeType.Paths:
		// Select path to read data from
		REPEAT
			iReadIndex := iReadIndex+1;
			IF (iReadIndex > MM_MAX_NUMBER_OF_PATH_ELEMENTS) THEN
				EXIT;
			END_IF
			UNTIL (abControlledPaths[i])
		END_REPEAT
		IF (iReadIndex <= MM_MAX_NUMBER_OF_PATH_ELEMENTS) THEN
			// Build remote symbol name
			sPrefix := CONCAT(sObjectIDentifier, '.stTrackStatus');
			// Data pointer for received data
			pReadNodeData := ADR(aReadPathData[iReadIndex]);
			// Header data size
			cbDataTotal := SIZEOF(aReadPathData[iReadIndex].stReadListReturnInfo);
			
			// Specify nodes to read by variable name
			nNoOfNodes := nNoOfNodes + 1;
			aNodeIDs[nNoOfNodes].sIdentifier := CONCAT(sPrefix, '.aPaths[');
			aNodeIDs[nNoOfNodes].sIdentifier := CONCAT(aNodeIDs[nNoOfNodes].sIdentifier, UINT_TO_STRING(iReadIndex));
			aNodeIDs[nNoOfNodes].sIdentifier := CONCAT(aNodeIDs[nNoOfNodes].sIdentifier, ']');
			acbDatas[nNoOfNodes] := SIZEOF(aReadPathData[iReadIndex]);
			cbDataTotal := cbDataTotal + acbDatas[nNoOfNodes];
			bReturn := TRUE;
		ELSE
			// Read next type
			iReadIndex := 0;
			eReadType := E_OPC_NodeType.Stations;
			bReturn := FALSE;
		END_IF
		
	E_OPC_NodeType.Stations:
		// Select Station to read data from
		iReadIndex := iReadIndex+1;
		IF (iReadIndex <= MM_MAX_NUMBER_OF_STATION_ELEMENTS) THEN
			// Build remote symbol name
			sPrefix := CONCAT(sObjectIDentifier, '.stTrackStatus');
			// Data pointer
			pReadNodeData := ADR(aReadStationData[iReadIndex]);
			
			// Header data
			cbDataTotal := SIZEOF(aReadStationData[iReadIndex].stReadListReturnInfo);
			
			// Specify nodes to read by variable name
			nNoOfNodes := nNoOfNodes + 1;
			aNodeIDs[nNoOfNodes].sIdentifier := CONCAT(sPrefix, '.aStations[');
			aNodeIDs[nNoOfNodes].sIdentifier := CONCAT(aNodeIDs[nNoOfNodes].sIdentifier, UINT_TO_STRING(iReadIndex));
			aNodeIDs[nNoOfNodes].sIdentifier := CONCAT(aNodeIDs[nNoOfNodes].sIdentifier, ']');
			acbDatas[nNoOfNodes] := SIZEOF(aReadStationData[iReadIndex].stStationData);
			cbDataTotal := cbDataTotal + acbDatas[nNoOfNodes];
			bReturn := TRUE;
		ELSE
			// Read next type
			iReadIndex := 0;
			eReadType := E_OPC_NodeType.Cells;
			bReturn := FALSE;
		END_IF
		
	E_OPC_NodeType.Cells:
		// Select cell status to read data from
		iReadIndex := iThisCellIndex;
		IF (iReadIndex > 0 AND iReadIndex <= MM_MAX_NUMBER_OF_STATION_ELEMENTS) THEN
			// Build remote symbol name
			sPrefix := CONCAT(sObjectIDentifier, '.stTrackStatus');
			// Data pointer
			pReadNodeData := ADR(aReadCellData);
			
			// Header data
			cbDataTotal := SIZEOF(aReadCellData.stReadListReturnInfo);
			
			// Specify nodes to read by variable name
			nNoOfNodes := nNoOfNodes + 1;
			aNodeIDs[nNoOfNodes].sIdentifier := CONCAT(sPrefix, '.aCells[');
			aNodeIDs[nNoOfNodes].sIdentifier := CONCAT(aNodeIDs[nNoOfNodes].sIdentifier, UINT_TO_STRING(iReadIndex));
			aNodeIDs[nNoOfNodes].sIdentifier := CONCAT(aNodeIDs[nNoOfNodes].sIdentifier, ']');
			acbDatas[nNoOfNodes] := SIZEOF(aReadCellData.stCell);
			cbDataTotal := cbDataTotal + acbDatas[nNoOfNodes]; 
			bReturn := TRUE;

			// continue to next type after this read!
			iReadIndex := 0;
			eReadType := E_OPC_NodeType.Vehicles;
		ELSE
			// Read next type
			iReadIndex := 0;
			eReadType := E_OPC_NodeType.Vehicles;
			bReturn := FALSE;
		END_IF
	
END_CASE
END_METHOD

METHOD PROTECTED M_InitNodeData_ADS : BOOL
VAR
	i				: UINT;
	sPrefix 		: STRING;
	
	bReturn			: BOOL;
END_VAR

nNoOfNodes := 0;
cbDataTotal := 0;

// TEST NEW
IF ( (nDecisionPointVehicleNo > 0) AND bReadDecPointVehicle ) THEN
	// Read data from vehicle at decision point (Higher priority!)
	// Build remote symbol name
	sPrefix := CONCAT(sObjectIDentifier, '.stTrackStatus');
	// Data pointer for received data
	pReadNodeData := ADR(aReadVehicleData[nDecisionPointVehicleNo].stVehicle);
	// Header data size
	cbDataTotal := SIZEOF(aReadVehicleData[nDecisionPointVehicleNo].stVehicle);
	
	// Specify nodes to read by variable name
	sTrackServerSymbol := CONCAT(sPrefix, '.aVehicles[');
	sTrackServerSymbol := CONCAT(sTrackServerSymbol, UINT_TO_STRING(nDecisionPointVehicleNo));
	sTrackServerSymbol := CONCAT(sTrackServerSymbol, ']');

	// Remove this vehicle from the event-driven reading list (to make sure it is not continously read!)
	M_VehicleToReadRemove(nDecisionPointVehicleNo);
				
	bReadDecPointVehicle := FALSE;	// Done in M_StateMachineNode_ADS
	bReadDecPointVehicleBusy := TRUE;
	bReturn := TRUE;

	M_InitNodeData_ADS := bReturn;
	RETURN;
END_IF
// END TEST NEW

// Comm type selection
CASE eReadType OF
	E_OPC_NodeType.Vehicles:
		IF ( (nDecisionPointVehicleNo > 0) AND bReadDecPointVehicle ) THEN
			// Read data from vehicle at decision point (Higher priority!)
			// Build remote symbol name
			sPrefix := CONCAT(sObjectIDentifier, '.stTrackStatus');
			// Data pointer for received data
			pReadNodeData := ADR(aReadVehicleData[nDecisionPointVehicleNo].stVehicle);
			// Header data size
			cbDataTotal := SIZEOF(aReadVehicleData[nDecisionPointVehicleNo].stVehicle);
			
			// Specify nodes to read by variable name
			sTrackServerSymbol := CONCAT(sPrefix, '.aVehicles[');
			sTrackServerSymbol := CONCAT(sTrackServerSymbol, UINT_TO_STRING(nDecisionPointVehicleNo));
			sTrackServerSymbol := CONCAT(sTrackServerSymbol, ']');

			// Remove this vehicle from the event-driven reading list (to make sure it is not continously read!)
			M_VehicleToReadRemove(nDecisionPointVehicleNo);
				
